LIN {X 0.166,Y -545.979,Z 599.154,A 0.000,B 0.000,C 90.000,E1 63.768} C_DIS
LIN {X 0.022,Y -541.378,Z 599.152,A 0.000,B 0.000,C 90.000,E1 63.435} C_DIS
LIN {X -0.133,Y -535.333,Z 599.150,A 0.000,B 0.000,C 90.000,E1 63.050} C_DIS
LIN {X 0.006,Y -529.277,Z 599.148,A 0.000,B 0.000,C 90.000,E1 62.666} C_DIS
LIN {X 0.118,Y -522.286,Z 599.146,A 0.000,B 0.000,C 90.000,E1 62.281} C_DIS
LIN {X -0.032,Y -515.785,Z 599.144,A 0.000,B 0.000,C 90.000,E1 61.975} C_DIS
LIN {X -0.104,Y -503.976,Z 599.141,A 0.000,B 0.000,C 90.000,E1 61.435} C_DIS
LIN {X -0.129,Y -485.175,Z 599.137,A 0.000,B 0.000,C 90.000,E1 60.589} C_DIS
LIN {X 0.140,Y -461.668,Z 599.130,A 0.000,B 0.000,C 90.000,E1 59.459} C_DIS
LIN {X 0.043,Y -448.327,Z 599.127,A 0.000,B 0.000,C 90.000,E1 58.791} C_DIS
LIN {X 0.001,Y -448.293,Z 599.127,A 0.000,B 0.000,C 90.000,E1 58.791} C_DIS
LIN {X -0.028,Y -444.314,Z 599.115,A 0.000,B 0.000,C 90.000,E1 56.707} C_DIS
LIN {X 0.030,Y -443.665,Z 599.113,A 0.000,B 0.000,C 90.000,E1 56.373} C_DIS
LIN {X 0.020,Y -434.553,Z 599.091,A 0.000,B 0.000,C 90.000,E1 52.431} C_DIS
LIN {X 0.117,Y -431.885,Z 599.083,A 0.000,B 0.000,C 90.000,E1 51.009} C_DIS
LIN {X 0.135,Y -433.279,Z 599.073,A 0.000,B 0.000,C 90.000,E1 49.094} C_DIS
LIN {X -0.208,Y -434.692,Z 599.062,A 0.000,B 0.000,C 90.000,E1 47.148} C_DIS
LIN {X -0.113,Y -435.635,Z 599.054,A 0.000,B 0.000,C 90.000,E1 45.810} C_DIS
LIN {X 0.205,Y -437.080,Z 599.043,A 0.000,B 0.000,C 90.000,E1 43.785} C_DIS
LIN {X 0.041,Y -437.949,Z 599.036,A 0.000,B 0.000,C 90.000,E1 42.486} C_DIS
LIN {X 0.186,Y -438.656,Z 599.029,A 0.000,B 0.000,C 90.000,E1 41.148} C_DIS
LIN {X 0.045,Y -439.277,Z 599.021,A 0.000,B 0.000,C 90.000,E1 39.850} C_DIS
LIN {X -0.061,Y -440.083,Z 599.010,A 0.000,B 0.000,C 90.000,E1 37.890} C_DIS
LIN {X -0.150,Y -440.627,Z 599.000,A 0.000,B 0.000,C 90.000,E1 35.931} C_DIS
LIN {X -0.066,Y -440.906,Z 598.990,A 0.000,B 0.000,C 90.000,E1 34.278} C_DIS
LIN {X -0.016,Y -441.048,Z 598.983,A 0.000,B 0.000,C 90.000,E1 32.959} C_DIS
LIN {X -0.206,Y -441.187,Z 598.976,A 0.000,B 0.000,C 90.000,E1 31.671} C_DIS
LIN {X 0.123,Y -441.488,Z 598.963,A 0.000,B 0.000,C 90.000,E1 29.333} C_DIS
LIN {X 0.016,Y -441.716,Z 598.950,A 0.000,B 0.000,C 90.000,E1 27.052} C_DIS
LIN {X 0.027,Y -441.984,Z 598.941,A 0.000,B 0.000,C 90.000,E1 25.412} C_DIS
LIN {X 0.052,Y -442.349,Z 598.932,A 0.000,B 0.000,C 90.000,E1 23.770} C_DIS
LIN {X -0.240,Y -442.753,Z 598.921,A 0.000,B 0.000,C 90.000,E1 21.844} C_DIS
LIN {X 0.023,Y -443.189,Z 598.912,A 0.000,B 0.000,C 90.000,E1 20.174} C_DIS
LIN {X 0.117,Y -443.894,Z 598.899,A 0.000,B 0.000,C 90.000,E1 17.873} C_DIS
LIN {X 0.242,Y -444.845,Z 598.885,A 0.000,B 0.000,C 90.000,E1 15.245} C_DIS
LIN {X 0.167,Y -446.065,Z 598.870,A 0.000,B 0.000,C 90.000,E1 12.647} C_DIS
LIN {X -0.067,Y -447.666,Z 598.856,A 0.000,B 0.000,C 90.000,E1 10.074} C_DIS
LIN {X -0.092,Y -448.788,Z 598.847,A 0.000,B 0.000,C 90.000,E1 8.454} C_DIS
LIN {X 0.101,Y -450.355,Z 598.836,A 0.000,B 0.000,C 90.000,E1 6.486} C_DIS
LIN {X 0.127,Y -452.695,Z 598.822,A 0.000,B 0.000,C 90.000,E1 3.898} C_DIS
LIN {X -0.197,Y -454.692,Z 598.811,A 0.000,B 0.000,C 90.000,E1 2.007} C_DIS
LIN {X -0.174,Y -458.491,Z 598.794,A 0.000,B 0.000,C 90.000,E1 358.854} C_DIS
LIN {X -0.200,Y -462.594,Z 598.778,A 0.000,B 0.000,C 90.000,E1 355.988} C_DIS
LIN {X 0.016,Y -465.061,Z 598.769,A 0.000,B 0.000,C 90.000,E1 354.375} C_DIS
LIN {X -0.162,Y -468.518,Z 598.757,A 0.000,B 0.000,C 90.000,E1 352.186} C_DIS
LIN {X 0.021,Y -470.459,Z 598.750,A 0.000,B 0.000,C 90.000,E1 350.905} C_DIS
LIN {X -0.186,Y -473.399,Z 598.739,A 0.000,B 0.000,C 90.000,E1 349.050} C_DIS
LIN {X 0.155,Y -477.086,Z 598.727,A 0.000,B 0.000,C 90.000,E1 346.825} C_DIS
LIN {X -0.079,Y -480.404,Z 598.717,A 0.000,B 0.000,C 90.000,E1 344.991} C_DIS
LIN {X -0.101,Y -483.276,Z 598.708,A 0.000,B 0.000,C 90.000,E1 343.449} C_DIS
LIN {X 0.073,Y -486.739,Z 598.698,A 0.000,B 0.000,C 90.000,E1 341.583} C_DIS
LIN {X -0.021,Y -489.139,Z 598.691,A 0.000,B 0.000,C 90.000,E1 340.369} C_DIS
LIN {X -0.049,Y -492.084,Z 598.682,A 0.000,B 0.000,C 90.000,E1 338.847} C_DIS
LIN {X 0.151,Y -494.806,Z 598.674,A 0.000,B 0.000,C 90.000,E1 337.305} C_DIS
LIN {X 0.145,Y -497.417,Z 598.666,A 0.000,B 0.000,C 90.000,E1 335.793} C_DIS
LIN {X -0.200,Y -500.222,Z 598.656,A 0.000,B 0.000,C 90.000,E1 334.024} C_DIS
LIN {X 0.050,Y -502.104,Z 598.649,A 0.000,B 0.000,C 90.000,E1 332.794} C_DIS
LIN {X -0.111,Y -505.249,Z 598.637,A 0.000,B 0.000,C 90.000,E1 330.717} C_DIS
LIN {X 0.042,Y -508.368,Z 598.626,A 0.000,B 0.000,C 90.000,E1 328.614} C_DIS
LIN {X -0.057,Y -511.830,Z 598.614,A 0.000,B 0.000,C 90.000,E1 326.548} C_DIS
LIN {X -0.129,Y -516.286,Z 598.601,A 0.000,B 0.000,C 90.000,E1 324.196} C_DIS
LIN {X -0.095,Y -519.677,Z 598.591,A 0.000,B 0.000,C 90.000,E1 322.431} C_DIS
LIN {X 0.243,Y -523.373,Z 598.582,A 0.000,B 0.000,C 90.000,E1 320.642} C_DIS
LIN {X 0.111,Y -525.794,Z 598.577,A 0.000,B 0.000,C 90.000,E1 319.784} C_DIS
LIN {X 0.011,Y -526.732,Z 598.575,A 0.000,B 0.000,C 90.000,E1 319.504} C_DIS
LIN {X 0.085,Y -529.285,Z 598.572,A 0.000,B 0.000,C 90.000,E1 318.933} C_DIS
LIN {X 0.244,Y -529.830,Z 598.571,A 0.000,B 0.000,C 90.000,E1 318.771} C_DIS
LIN {X 0.215,Y -531.524,Z 598.570,A 0.000,B 0.000,C 90.000,E1 318.485} C_DIS
LIN {X -0.144,Y -534.100,Z 598.568,A 0.000,B 0.000,C 90.000,E1 318.243} C_DIS
LIN {X -0.100,Y -536.720,Z 598.566,A 0.000,B 0.000,C 90.000,E1 317.957} C_DIS
LIN {X -0.059,Y -539.484,Z 598.565,A 0.000,B 0.000,C 90.000,E1 317.676} C_DIS
LIN {X -0.062,Y -544.568,Z 598.562,A 0.000,B 0.000,C 90.000,E1 317.229} C_DIS
LIN {X 0.172,Y -566.738,Z 598.553,A 0.000,B 0.000,C 90.000,E1 315.486} C_DIS
LIN {X -0.044,Y -584.428,Z 598.546,A 0.000,B 0.000,C 90.000,E1 314.190} C_DIS
LIN {X -0.296,Y -590.237,Z 598.543,A 0.000,B 0.000,C 90.000,E1 313.785} C_DIS
LIN {X -0.116,Y -598.732,Z 598.539,A 0.000,B 0.000,C 90.000,E1 313.095} C_DIS
LIN {X 0.176,Y -604.081,Z 598.537,A 0.000,B 0.000,C 90.000,E1 312.609} C_DIS
LIN {X -0.228,Y -608.017,Z 598.535,A 0.000,B 0.000,C 90.000,E1 312.285} C_DIS
LIN {X -0.022,Y -616.798,Z 598.530,A 0.000,B 0.000,C 90.000,E1 311.391} C_DIS
LIN {X -0.281,Y -624.670,Z 598.525,A 0.000,B 0.000,C 90.000,E1 310.539} C_DIS
LIN {X 0.259,Y -631.210,Z 598.521,A 0.000,B 0.000,C 90.000,E1 309.725} C_DIS
LIN {X 0.001,Y -637.456,Z 598.517,A 0.000,B 0.000,C 90.000,E1 308.991} C_DIS
LIN {X 0.184,Y -644.336,Z 598.512,A 0.000,B 0.000,C 90.000,E1 308.096} C_DIS
LIN {X -0.383,Y -648.858,Z 598.508,A 0.000,B 0.000,C 90.000,E1 307.523} C_DIS
LIN {X -0.030,Y -652.251,Z 598.506,A 0.000,B 0.000,C 90.000,E1 306.996} C_DIS
LIN {X -0.048,Y -655.376,Z 598.503,A 0.000,B 0.000,C 90.000,E1 306.503} C_DIS
LIN {X -0.004,Y -658.863,Z 598.499,A 0.000,B 0.000,C 90.000,E1 305.884} C_DIS
LIN {X 0.077,Y -662.080,Z 598.496,A 0.000,B 0.000,C 90.000,E1 305.264} C_DIS
LIN {X 0.074,Y -663.896,Z 598.494,A 0.000,B 0.000,C 90.000,E1 304.898} C_DIS
LIN {X -0.295,Y -667.172,Z 598.490,A 0.000,B 0.000,C 90.000,E1 304.199} C_DIS
LIN {X -0.080,Y -670.198,Z 598.486,A 0.000,B 0.000,C 90.000,E1 303.452} C_DIS
LIN {X -0.396,Y -672.978,Z 598.482,A 0.000,B 0.000,C 90.000,E1 302.752} C_DIS
LIN {X -0.001,Y -677.459,Z 598.475,A 0.000,B 0.000,C 90.000,E1 301.514} C_DIS
LIN {X -0.040,Y -682.613,Z 598.467,A 0.000,B 0.000,C 90.000,E1 300.079} C_DIS
LIN {X -0.063,Y -685.873,Z 598.462,A 0.000,B 0.000,C 90.000,E1 299.127} C_DIS
LIN {X 0.214,Y -688.976,Z 598.457,A 0.000,B 0.000,C 90.000,E1 298.153} C_DIS
LIN {X 0.217,Y -691.869,Z 598.451,A 0.000,B 0.000,C 90.000,E1 297.206} C_DIS
LIN {X 0.084,Y -693.221,Z 598.449,A 0.000,B 0.000,C 90.000,E1 296.744} C_DIS
LIN {X -0.045,Y -694.071,Z 598.446,A 0.000,B 0.000,C 90.000,E1 296.283} C_DIS
LIN {X -0.102,Y -694.440,Z 598.445,A 0.000,B 0.000,C 90.000,E1 296.052} C_DIS
LIN {X 0.149,Y -694.357,Z 598.443,A 0.000,B 0.000,C 90.000,E1 295.796} C_DIS
LIN {X 0.025,Y -693.740,Z 598.441,A 0.000,B 0.000,C 90.000,E1 295.335} C_DIS
LIN {X 0.273,Y -692.734,Z 598.440,A 0.000,B 0.000,C 90.000,E1 295.079} C_DIS
LIN {X -0.278,Y -690.914,Z 598.438,A 0.000,B 0.000,C 90.000,E1 294.771} C_DIS
LIN {X -0.158,Y -690.215,Z 598.437,A 0.000,B 0.000,C 90.000,E1 294.643} C_DIS
LIN {X -0.039,Y -689.136,Z 598.436,A 0.000,B 0.000,C 90.000,E1 294.515} C_DIS
LIN {X 0.078,Y -687.455,Z 598.436,A 0.000,B 0.000,C 90.000,E1 294.387} C_DIS
LIN {X -0.137,Y -683.985,Z 598.434,A 0.000,B 0.000,C 90.000,E1 294.207} C_DIS
LIN {X -0.111,Y -682.117,Z 598.434,A 0.000,B 0.000,C 90.000,E1 294.079} C_DIS
LIN {X 0.259,Y -680.132,Z 598.433,A 0.000,B 0.000,C 90.000,E1 293.951} C_DIS
LIN {X -0.069,Y -673.321,Z 598.432,A 0.000,B 0.000,C 90.000,E1 293.770} C_DIS
LIN {X 0.235,Y -669.043,Z 598.432,A 0.000,B 0.000,C 90.000,E1 293.643} C_DIS
LIN {X -0.119,Y -659.386,Z 598.431,A 0.000,B 0.000,C 90.000,E1 293.515} C_DIS
LIN {X -0.084,Y -646.367,Z 598.430,A 0.000,B 0.000,C 90.000,E1 293.334} C_DIS
LIN {X -0.034,Y -636.744,Z 598.429,A 0.000,B 0.000,C 90.000,E1 293.153} C_DIS
LIN {X -0.173,Y -627.009,Z 598.427,A 0.000,B 0.000,C 90.000,E1 292.950} C_DIS
LIN {X -0.121,Y -613.924,Z 598.425,A 0.000,B 0.000,C 90.000,E1 292.589} C_DIS
LIN {X 0.130,Y -579.349,Z 598.419,A 0.000,B 0.000,C 90.000,E1 291.482} C_DIS
LIN {X 0.137,Y -569.347,Z 598.418,A 0.000,B 0.000,C 90.000,E1 291.173} C_DIS
LIN {X -0.267,Y -565.886,Z 598.417,A 0.000,B 0.000,C 90.000,E1 291.099} C_DIS
LIN {X -0.154,Y -563.479,Z 598.416,A 0.000,B 0.000,C 90.000,E1 290.972} C_DIS
LIN {X 0.119,Y -560.661,Z 598.416,A 0.000,B 0.000,C 90.000,E1 290.791} C_DIS
LIN {X 0.065,Y -560.619,Z 598.416,A 0.000,B 0.000,C 90.000,E1 290.791} C_DIS
LIN {X -0.201,Y -559.519,Z 598.415,A 0.000,B 0.000,C 90.000,E1 290.663} C_DIS
LIN {X 0.279,Y -559.491,Z 598.415,A 0.000,B 0.000,C 90.000,E1 290.610} C_DIS
LIN {X -0.199,Y -558.876,Z 598.412,A 0.000,B 0.000,C 90.000,E1 290.248} C_DIS
LIN {X 0.055,Y -558.699,Z 598.402,A 0.000,B 0.000,C 90.000,E1 288.362} C_DIS
LIN {X 0.240,Y -558.547,Z 598.397,A 0.000,B 0.000,C 90.000,E1 287.511} C_DIS
LIN {X 0.137,Y -558.104,Z 598.390,A 0.000,B 0.000,C 90.000,E1 286.134} C_DIS
LIN {X 0.279,Y -557.667,Z 598.384,A 0.000,B 0.000,C 90.000,E1 285.009} C_DIS
LIN {X 0.145,Y -556.814,Z 598.374,A 0.000,B 0.000,C 90.000,E1 283.355} C_DIS
LIN {X -0.265,Y -556.046,Z 598.367,A 0.000,B 0.000,C 90.000,E1 282.007} C_DIS
LIN {X 0.115,Y -554.956,Z 598.356,A 0.000,B 0.000,C 90.000,E1 280.018} C_DIS
LIN {X -0.275,Y -553.920,Z 598.345,A 0.000,B 0.000,C 90.000,E1 278.106} C_DIS
LIN {X 0.177,Y -553.280,Z 598.337,A 0.000,B 0.000,C 90.000,E1 276.663} C_DIS
LIN {X 0.118,Y -552.541,Z 598.328,A 0.000,B 0.000,C 90.000,E1 274.992} C_DIS
LIN {X 0.088,Y -551.894,Z 598.317,A 0.000,B 0.000,C 90.000,E1 273.037} C_DIS
LIN {X -0.023,Y -551.381,Z 598.306,A 0.000,B 0.000,C 90.000,E1 271.088} C_DIS
LIN {X -0.271,Y -551.012,Z 598.298,A 0.000,B 0.000,C 90.000,E1 269.714} C_DIS
LIN {X 0.153,Y -550.278,Z 598.287,A 0.000,B 0.000,C 90.000,E1 267.707} C_DIS
LIN {X -0.102,Y -549.713,Z 598.280,A 0.000,B 0.000,C 90.000,E1 266.331} C_DIS
LIN {X 0.215,Y -549.027,Z 598.272,A 0.000,B 0.000,C 90.000,E1 264.894} C_DIS
LIN {X -0.033,Y -548.223,Z 598.264,A 0.000,B 0.000,C 90.000,E1 263.514} C_DIS
LIN {X 0.281,Y -547.287,Z 598.258,A 0.000,B 0.000,C 90.000,E1 262.356} C_DIS
LIN {X 0.058,Y -546.050,Z 598.250,A 0.000,B 0.000,C 90.000,E1 260.971} C_DIS
LIN {X 0.068,Y -544.125,Z 598.239,A 0.000,B 0.000,C 90.000,E1 258.993} C_DIS
LIN {X -0.115,Y -543.093,Z 598.233,A 0.000,B 0.000,C 90.000,E1 257.881} C_DIS
LIN {X -0.033,Y -541.350,Z 598.223,A 0.000,B 0.000,C 90.000,E1 256.172} C_DIS
LIN {X -0.128,Y -540.226,Z 598.217,A 0.000,B 0.000,C 90.000,E1 255.046} C_DIS
LIN {X -0.027,Y -538.775,Z 598.209,A 0.000,B 0.000,C 90.000,E1 253.614} C_DIS
LIN {X 0.045,Y -537.283,Z 598.201,A 0.000,B 0.000,C 90.000,E1 252.181} C_DIS
LIN {X 0.038,Y -536.067,Z 598.195,A 0.000,B 0.000,C 90.000,E1 251.040} C_DIS
LIN {X -0.109,Y -534.119,Z 598.187,A 0.000,B 0.000,C 90.000,E1 249.625} C_DIS
LIN {X 0.213,Y -531.664,Z 598.179,A 0.000,B 0.000,C 90.000,E1 248.156} C_DIS
LIN {X -0.199,Y -529.517,Z 598.172,A 0.000,B 0.000,C 90.000,E1 247.050} C_DIS
LIN {X -0.261,Y -526.695,Z 598.164,A 0.000,B 0.000,C 90.000,E1 245.613} C_DIS
LIN {X -0.155,Y -523.732,Z 598.156,A 0.000,B 0.000,C 90.000,E1 244.152} C_DIS
LIN {X 0.130,Y -520.515,Z 598.148,A 0.000,B 0.000,C 90.000,E1 242.666} C_DIS
LIN {X -0.014,Y -517.839,Z 598.142,A 0.000,B 0.000,C 90.000,E1 241.513} C_DIS
LIN {X 0.044,Y -514.913,Z 598.135,A 0.000,B 0.000,C 90.000,E1 240.333} C_DIS
LIN {X -0.153,Y -509.069,Z 598.122,A 0.000,B 0.000,C 90.000,E1 237.995} C_DIS
LIN {X 0.028,Y -506.047,Z 598.116,A 0.000,B 0.000,C 90.000,E1 236.786} C_DIS
LIN {X 0.018,Y -502.654,Z 598.109,A 0.000,B 0.000,C 90.000,E1 235.595} C_DIS
LIN {X -0.034,Y -499.205,Z 598.102,A 0.000,B 0.000,C 90.000,E1 234.402} C_DIS
LIN {X -0.152,Y -491.971,Z 598.087,A 0.000,B 0.000,C 90.000,E1 231.698} C_DIS
LIN {X 0.068,Y -487.986,Z 598.079,A 0.000,B 0.000,C 90.000,E1 230.150} C_DIS
LIN {X 0.015,Y -484.808,Z 598.072,A 0.000,B 0.000,C 90.000,E1 228.933} C_DIS
LIN {X -0.028,Y -479.413,Z 598.060,A 0.000,B 0.000,C 90.000,E1 226.782} C_DIS
LIN {X -0.009,Y -474.908,Z 598.050,A 0.000,B 0.000,C 90.000,E1 224.919} C_DIS
LIN {X -0.181,Y -471.290,Z 598.041,A 0.000,B 0.000,C 90.000,E1 223.380} C_DIS
LIN {X 0.021,Y -466.931,Z 598.030,A 0.000,B 0.000,C 90.000,E1 221.472} C_DIS
LIN {X -0.034,Y -464.181,Z 598.023,A 0.000,B 0.000,C 90.000,E1 220.216} C_DIS
LIN {X -0.203,Y -459.497,Z 598.011,A 0.000,B 0.000,C 90.000,E1 218.016} C_DIS
LIN {X 0.035,Y -456.868,Z 598.004,A 0.000,B 0.000,C 90.000,E1 216.710} C_DIS
LIN {X 0.052,Y -453.745,Z 597.995,A 0.000,B 0.000,C 90.000,E1 215.105} C_DIS
LIN {X -0.116,Y -448.841,Z 597.981,A 0.000,B 0.000,C 90.000,E1 212.546} C_DIS
LIN {X -0.054,Y -445.372,Z 597.970,A 0.000,B 0.000,C 90.000,E1 210.590} C_DIS
LIN {X 0.079,Y -441.814,Z 597.959,A 0.000,B 0.000,C 90.000,E1 208.615} C_DIS
LIN {X -0.084,Y -438.365,Z 597.948,A 0.000,B 0.000,C 90.000,E1 206.668} C_DIS
LIN {X -0.149,Y -435.482,Z 597.939,A 0.000,B 0.000,C 90.000,E1 205.027} C_DIS
LIN {X -0.047,Y -432.098,Z 597.928,A 0.000,B 0.000,C 90.000,E1 203.025} C_DIS
LIN {X 0.000,Y -429.390,Z 597.919,A 0.000,B 0.000,C 90.000,E1 201.354} C_DIS
LIN {X -0.162,Y -425.683,Z 597.906,A 0.000,B 0.000,C 90.000,E1 199.033} C_DIS
LIN {X 0.056,Y -422.755,Z 597.894,A 0.000,B 0.000,C 90.000,E1 196.985} C_DIS
LIN {X 0.075,Y -419.965,Z 597.883,A 0.000,B 0.000,C 90.000,E1 194.954} C_DIS
LIN {X 0.111,Y -418.085,Z 597.876,A 0.000,B 0.000,C 90.000,E1 193.592} C_DIS
LIN {X 0.204,Y -415.072,Z 597.864,A 0.000,B 0.000,C 90.000,E1 191.535} C_DIS
LIN {X 0.176,Y -410.918,Z 597.847,A 0.000,B 0.000,C 90.000,E1 188.454} C_DIS
LIN {X -0.144,Y -408.830,Z 597.838,A 0.000,B 0.000,C 90.000,E1 186.777} C_DIS
LIN {X -0.168,Y -405.709,Z 597.824,A 0.000,B 0.000,C 90.000,E1 184.359} C_DIS
LIN {X -0.135,Y -401.282,Z 597.799,A 0.000,B 0.000,C 90.000,E1 179.828} C_DIS
LIN {X -0.112,Y -399.169,Z 597.781,A 0.000,B 0.000,C 90.000,E1 176.674} C_DIS
LIN {X -0.051,Y -398.035,Z 597.766,A 0.000,B 0.000,C 90.000,E1 173.856} C_DIS
LIN {X 0.078,Y -397.457,Z 597.752,A 0.000,B 0.000,C 90.000,E1 171.376} C_DIS
LIN {X -0.044,Y -397.250,Z 597.737,A 0.000,B 0.000,C 90.000,E1 168.578} C_DIS
LIN {X 0.002,Y -397.566,Z 597.721,A 0.000,B 0.000,C 90.000,E1 165.755} C_DIS
LIN {X 0.104,Y -398.040,Z 597.709,A 0.000,B 0.000,C 90.000,E1 163.630} C_DIS
LIN {X 0.099,Y -398.630,Z 597.699,A 0.000,B 0.000,C 90.000,E1 161.873} C_DIS
LIN {X -0.099,Y -399.432,Z 597.686,A 0.000,B 0.000,C 90.000,E1 159.444} C_DIS
LIN {X -0.225,Y -400.269,Z 597.674,A 0.000,B 0.000,C 90.000,E1 157.358} C_DIS
LIN {X -0.026,Y -401.172,Z 597.662,A 0.000,B 0.000,C 90.000,E1 155.229} C_DIS
LIN {X 0.114,Y -401.924,Z 597.653,A 0.000,B 0.000,C 90.000,E1 153.461} C_DIS
LIN {X -0.161,Y -402.572,Z 597.645,A 0.000,B 0.000,C 90.000,E1 152.103} C_DIS
LIN {X -0.086,Y -403.408,Z 597.633,A 0.000,B 0.000,C 90.000,E1 149.999} C_DIS
LIN {X -0.033,Y -403.993,Z 597.624,A 0.000,B 0.000,C 90.000,E1 148.250} C_DIS
LIN {X 0.030,Y -404.457,Z 597.614,A 0.000,B 0.000,C 90.000,E1 146.501} C_DIS
LIN {X 0.111,Y -404.966,Z 597.602,A 0.000,B 0.000,C 90.000,E1 144.402} C_DIS
LIN {X -0.126,Y -405.515,Z 597.591,A 0.000,B 0.000,C 90.000,E1 142.351} C_DIS
LIN {X -0.175,Y -406.136,Z 597.579,A 0.000,B 0.000,C 90.000,E1 140.275} C_DIS
LIN {X 0.053,Y -406.672,Z 597.568,A 0.000,B 0.000,C 90.000,E1 138.162} C_DIS
LIN {X 0.005,Y -406.892,Z 597.560,A 0.000,B 0.000,C 90.000,E1 136.782} C_DIS
LIN {X 0.204,Y -407.210,Z 597.548,A 0.000,B 0.000,C 90.000,E1 134.676} C_DIS
LIN {X -0.011,Y -407.436,Z 597.539,A 0.000,B 0.000,C 90.000,E1 132.975} C_DIS
LIN {X -0.065,Y -407.624,Z 597.527,A 0.000,B 0.000,C 90.000,E1 130.906} C_DIS
LIN {X -0.215,Y -407.826,Z 597.518,A 0.000,B 0.000,C 90.000,E1 129.197} C_DIS
LIN {X -0.151,Y -407.834,Z 597.515,A 0.000,B 0.000,C 90.000,E1 128.669} C_DIS
LIN {X -0.201,Y -415.250,Z 597.500,A 0.000,B 0.000,C 90.000,E1 126.091} C_DIS
LIN {X -0.091,Y -416.909,Z 597.497,A 0.000,B 0.000,C 90.000,E1 125.391} C_DIS
LIN {X 0.101,Y -425.710,Z 597.478,A 0.000,B 0.000,C 90.000,E1 121.957} C_DIS
LIN {X 0.062,Y -425.748,Z 597.478,A 0.000,B 0.000,C 90.000,E1 121.957} C_DIS
LIN {X 0.143,Y -435.597,Z 597.475,A 0.000,B 0.000,C 90.000,E1 121.465} C_DIS
LIN {X -0.037,Y -442.412,Z 597.473,A 0.000,B 0.000,C 90.000,E1 121.180} C_DIS
LIN {X -0.064,Y -449.171,Z 597.471,A 0.000,B 0.000,C 90.000,E1 120.846} C_DIS
LIN {X 0.070,Y -452.676,Z 597.470,A 0.000,B 0.000,C 90.000,E1 120.669} C_DIS
LIN {X 0.030,Y -466.023,Z 597.467,A 0.000,B 0.000,C 90.000,E1 120.001} C_DIS
LIN {X 0.058,Y -475.942,Z 597.464,A 0.000,B 0.000,C 90.000,E1 119.461} C_DIS
LIN {X 0.201,Y -482.620,Z 597.462,A 0.000,B 0.000,C 90.000,E1 119.077} C_DIS
LIN {X -0.146,Y -493.965,Z 597.458,A 0.000,B 0.000,C 90.000,E1 118.437} C_DIS
LIN {X -0.083,Y -500.278,Z 597.456,A 0.000,B 0.000,C 90.000,E1 118.025} C_DIS
LIN {X 0.037,Y -509.700,Z 597.452,A 0.000,B 0.000,C 90.000,E1 117.385} C_DIS
LIN {X -0.148,Y -519.934,Z 597.448,A 0.000,B 0.000,C 90.000,E1 116.668} C_DIS
LIN {X -0.032,Y -527.143,Z 597.445,A 0.000,B 0.000,C 90.000,E1 116.104} C_DIS
LIN {X -0.109,Y -532.984,Z 597.442,A 0.000,B 0.000,C 90.000,E1 115.643} C_DIS
LIN {X 0.040,Y -540.321,Z 597.439,A 0.000,B 0.000,C 90.000,E1 115.027} C_DIS
LIN {X 0.195,Y -545.812,Z 597.436,A 0.000,B 0.000,C 90.000,E1 114.515} C_DIS
LIN {X -0.133,Y -550.789,Z 597.434,A 0.000,B 0.000,C 90.000,E1 114.079} C_DIS
LIN {X -0.126,Y -555.397,Z 597.431,A 0.000,B 0.000,C 90.000,E1 113.567} C_DIS
LIN {X 0.171,Y -561.281,Z 597.427,A 0.000,B 0.000,C 90.000,E1 112.823} C_DIS
LIN {X -0.257,Y -563.091,Z 597.425,A 0.000,B 0.000,C 90.000,E1 112.589} C_DIS
LIN {X -0.168,Y -565.816,Z 597.423,A 0.000,B 0.000,C 90.000,E1 112.206} C_DIS
LIN {X -0.336,Y -570.004,Z 597.419,A 0.000,B 0.000,C 90.000,E1 111.535} C_DIS
LIN {X 0.190,Y -574.425,Z 597.415,A 0.000,B 0.000,C 90.000,E1 110.663} C_DIS
LIN {X -0.178,Y -578.433,Z 597.410,A 0.000,B 0.000,C 90.000,E1 109.885} C_DIS
LIN {X 0.042,Y -580.900,Z 597.407,A 0.000,B 0.000,C 90.000,E1 109.322} C_DIS
LIN {X -0.259,Y -584.375,Z 597.403,A 0.000,B 0.000,C 90.000,E1 108.544} C_DIS
LIN {X -0.194,Y -586.556,Z 597.400,A 0.000,B 0.000,C 90.000,E1 108.000} C_DIS
LIN {X -0.021,Y -590.310,Z 597.394,A 0.000,B 0.000,C 90.000,E1 106.913} C_DIS
LIN {X -0.229,Y -592.947,Z 597.390,A 0.000,B 0.000,C 90.000,E1 106.134} C_DIS
LIN {X 0.138,Y -597.029,Z 597.382,A 0.000,B 0.000,C 90.000,E1 104.773} C_DIS
LIN {X 0.301,Y -602.058,Z 597.373,A 0.000,B 0.000,C 90.000,E1 103.175} C_DIS
LIN {X 0.041,Y -607.979,Z 597.363,A 0.000,B 0.000,C 90.000,E1 101.366} C_DIS
LIN {X -0.064,Y -612.191,Z 597.356,A 0.000,B 0.000,C 90.000,E1 100.074} C_DIS
LIN {X -0.315,Y -616.167,Z 597.349,A 0.000,B 0.000,C 90.000,E1 98.803} C_DIS
LIN {X 0.124,Y -619.932,Z 597.342,A 0.000,B 0.000,C 90.000,E1 97.473} C_DIS
LIN {X 0.011,Y -623.481,Z 597.335,A 0.000,B 0.000,C 90.000,E1 96.201} C_DIS
LIN {X -0.148,Y -625.431,Z 597.330,A 0.000,B 0.000,C 90.000,E1 95.448} C_DIS
LIN {X 0.273,Y -627.230,Z 597.326,A 0.000,B 0.000,C 90.000,E1 94.645} C_DIS
LIN {X 0.090,Y -628.750,Z 597.322,A 0.000,B 0.000,C 90.000,E1 93.898} C_DIS
LIN {X 0.273,Y -630.629,Z 597.316,A 0.000,B 0.000,C 90.000,E1 92.865} C_DIS
LIN {X 0.213,Y -632.546,Z 597.309,A 0.000,B 0.000,C 90.000,E1 91.604} C_DIS
LIN {X 0.056,Y -633.540,Z 597.305,A 0.000,B 0.000,C 90.000,E1 90.859} C_DIS
LIN {X -0.090,Y -634.288,Z 597.301,A 0.000,B 0.000,C 90.000,E1 90.115} C_DIS
LIN {X -0.226,Y -634.788,Z 597.296,A 0.000,B 0.000,C 90.000,E1 89.370} C_DIS
LIN {X 0.274,Y -635.067,Z 597.292,A 0.000,B 0.000,C 90.000,E1 88.568} C_DIS
LIN {X 0.162,Y -635.153,Z 597.288,A 0.000,B 0.000,C 90.000,E1 87.822} C_DIS
LIN {X -0.199,Y -634.893,Z 597.282,A 0.000,B 0.000,C 90.000,E1 86.846} C_DIS
LIN {X 0.288,Y -634.496,Z 597.278,A 0.000,B 0.000,C 90.000,E1 86.045} C_DIS
LIN {X -0.039,Y -633.735,Z 597.273,A 0.000,B 0.000,C 90.000,E1 85.065} C_DIS
LIN {X -0.008,Y -632.447,Z 597.266,A 0.000,B 0.000,C 90.000,E1 83.799} C_DIS
LIN {X 0.138,Y -631.854,Z 597.263,A 0.000,B 0.000,C 90.000,E1 83.280} C_DIS
LIN {X -0.010,Y -630.674,Z 597.259,A 0.000,B 0.000,C 90.000,E1 82.534} C_DIS
LIN {X -0.294,Y -628.902,Z 597.253,A 0.000,B 0.000,C 90.000,E1 81.546} C_DIS
LIN {X 0.234,Y -627.372,Z 597.249,A 0.000,B 0.000,C 90.000,E1 80.735} C_DIS
LIN {X 0.320,Y -624.623,Z 597.242,A 0.000,B 0.000,C 90.000,E1 79.454} C_DIS
LIN {X -0.254,Y -621.558,Z 597.235,A 0.000,B 0.000,C 90.000,E1 78.229} C_DIS
LIN {X 0.082,Y -618.908,Z 597.229,A 0.000,B 0.000,C 90.000,E1 77.173} C_DIS
LIN {X -0.222,Y -616.052,Z 597.223,A 0.000,B 0.000,C 90.000,E1 76.172} C_DIS
LIN {X -0.056,Y -612.192,Z 597.216,A 0.000,B 0.000,C 90.000,E1 74.866} C_DIS
LIN {X -0.204,Y -609.669,Z 597.212,A 0.000,B 0.000,C 90.000,E1 74.102} C_DIS
LIN {X -0.214,Y -606.897,Z 597.207,A 0.000,B 0.000,C 90.000,E1 73.323} C_DIS
LIN {X -0.251,Y -603.838,Z 597.203,A 0.000,B 0.000,C 90.000,E1 72.543} C_DIS
LIN {X -0.319,Y -600.529,Z 597.199,A 0.000,B 0.000,C 90.000,E1 71.764} C_DIS
LIN {X -0.180,Y -597.576,Z 597.195,A 0.000,B 0.000,C 90.000,E1 71.094} C_DIS
LIN {X -0.122,Y -593.748,Z 597.190,A 0.000,B 0.000,C 90.000,E1 70.296} C_DIS
LIN {X -0.043,Y -590.353,Z 597.187,A 0.000,B 0.000,C 90.000,E1 69.625} C_DIS
LIN {X 0.004,Y -586.670,Z 597.183,A 0.000,B 0.000,C 90.000,E1 68.954} C_DIS
LIN {X 0.055,Y -582.749,Z 597.179,A 0.000,B 0.000,C 90.000,E1 68.284} C_DIS
LIN {X -0.263,Y -579.534,Z 597.177,A 0.000,B 0.000,C 90.000,E1 67.794} C_DIS
LIN {X 0.086,Y -574.070,Z 597.172,A 0.000,B 0.000,C 90.000,E1 66.975} C_DIS
LIN {X -0.201,Y -570.192,Z 597.169,A 0.000,B 0.000,C 90.000,E1 66.485} C_DIS
LIN {X 0.253,Y -564.781,Z 597.166,A 0.000,B 0.000,C 90.000,E1 65.793} C_DIS
LIN {X 0.097,Y -560.305,Z 597.163,A 0.000,B 0.000,C 90.000,E1 65.305} C_DIS
LIN {X -0.252,Y -555.562,Z 597.160,A 0.000,B 0.000,C 90.000,E1 64.845} C_DIS
LIN {X 0.046,Y -550.417,Z 597.157,A 0.000,B 0.000,C 90.000,E1 64.332} C_DIS
LIN {X -0.183,Y -544.861,Z 597.155,A 0.000,B 0.000,C 90.000,E1 63.896} C_DIS
LIN {X -0.032,Y -539.093,Z 597.153,A 0.000,B 0.000,C 90.000,E1 63.461} C_DIS
LIN {X 0.178,Y -534.164,Z 597.151,A 0.000,B 0.000,C 90.000,E1 63.127} C_DIS
LIN {X 0.192,Y -527.618,Z 597.149,A 0.000,B 0.000,C 90.000,E1 62.743} C_DIS
LIN {X -0.099,Y -520.593,Z 597.147,A 0.000,B 0.000,C 90.000,E1 62.410} C_DIS
LIN {X -0.050,Y -515.458,Z 597.145,A 0.000,B 0.000,C 90.000,E1 62.153} C_DIS
LIN {X 0.023,Y -503.311,Z 597.142,A 0.000,B 0.000,C 90.000,E1 61.591} C_DIS
LIN {X 0.072,Y -482.856,Z 597.137,A 0.000,B 0.000,C 90.000,E1 60.667} C_DIS
LIN {X -0.103,Y -462.472,Z 597.132,A 0.000,B 0.000,C 90.000,E1 59.744} C_DIS
LIN {X -0.278,Y -448.859,Z 597.128,A 0.000,B 0.000,C 90.000,E1 59.076} C_DIS
LIN {X 0.295,Y -448.803,Z 597.128,A 0.000,B 0.000,C 90.000,E1 58.997} C_DIS
LIN {X 0.138,Y -444.131,Z 597.115,A 0.000,B 0.000,C 90.000,E1 56.580} C_DIS
LIN {X 0.128,Y -442.543,Z 597.111,A 0.000,B 0.000,C 90.000,E1 55.928} C_DIS
LIN {X 0.084,Y -433.691,Z 597.089,A 0.000,B 0.000,C 90.000,E1 51.984} C_DIS
LIN {X -0.012,Y -432.290,Z 597.085,A 0.000,B 0.000,C 90.000,E1 51.251} C_DIS
LIN {X 0.190,Y -432.649,Z 597.082,A 0.000,B 0.000,C 90.000,E1 50.642} C_DIS
LIN {X -0.058,Y -433.941,Z 597.072,A 0.000,B 0.000,C 90.000,E1 49.013} C_DIS
LIN {X 0.286,Y -435.162,Z 597.063,A 0.000,B 0.000,C 90.000,E1 47.310} C_DIS
LIN {X -0.228,Y -436.185,Z 597.056,A 0.000,B 0.000,C 90.000,E1 46.053} C_DIS
LIN {X 0.057,Y -437.911,Z 597.043,A 0.000,B 0.000,C 90.000,E1 43.704} C_DIS
LIN {X 0.201,Y -438.752,Z 597.036,A 0.000,B 0.000,C 90.000,E1 42.366} C_DIS
LIN {X 0.063,Y -439.459,Z 597.028,A 0.000,B 0.000,C 90.000,E1 41.067} C_DIS
LIN {X -0.068,Y -440.051,Z 597.021,A 0.000,B 0.000,C 90.000,E1 39.769} C_DIS
LIN {X -0.158,Y -440.829,Z 597.010,A 0.000,B 0.000,C 90.000,E1 37.810} C_DIS
LIN {X -0.172,Y -441.252,Z 597.001,A 0.000,B 0.000,C 90.000,E1 36.171} C_DIS
LIN {X -0.182,Y -441.548,Z 596.992,A 0.000,B 0.000,C 90.000,E1 34.532} C_DIS
LIN {X -0.126,Y -441.643,Z 596.984,A 0.000,B 0.000,C 90.000,E1 33.214} C_DIS
LIN {X 0.113,Y -441.805,Z 596.975,A 0.000,B 0.000,C 90.000,E1 31.544} C_DIS
LIN {X 0.028,Y -441.995,Z 596.964,A 0.000,B 0.000,C 90.000,E1 29.589} C_DIS
LIN {X -0.067,Y -442.208,Z 596.952,A 0.000,B 0.000,C 90.000,E1 27.308} C_DIS
LIN {X -0.009,Y -442.480,Z 596.941,A 0.000,B 0.000,C 90.000,E1 25.335} C_DIS
LIN {X 0.019,Y -442.801,Z 596.932,A 0.000,B 0.000,C 90.000,E1 23.695} C_DIS
LIN {X -0.125,Y -443.125,Z 596.923,A 0.000,B 0.000,C 90.000,E1 22.078} C_DIS
LIN {X -0.015,Y -443.531,Z 596.914,A 0.000,B 0.000,C 90.000,E1 20.429} C_DIS
LIN {X -0.048,Y -444.240,Z 596.899,A 0.000,B 0.000,C 90.000,E1 17.819} C_DIS
LIN {X -0.183,Y -445.047,Z 596.886,A 0.000,B 0.000,C 90.000,E1 15.552} C_DIS
LIN {X -0.140,Y -446.219,Z 596.872,A 0.000,B 0.000,C 90.000,E1 12.939} C_DIS
LIN {X 0.068,Y -447.747,Z 596.857,A 0.000,B 0.000,C 90.000,E1 10.310} C_DIS
LIN {X 0.117,Y -448.854,Z 596.848,A 0.000,B 0.000,C 90.000,E1 8.681} C_DIS
LIN {X -0.004,Y -450.610,Z 596.836,A 0.000,B 0.000,C 90.000,E1 6.429} C_DIS
LIN {X -0.163,Y -452.637,Z 596.823,A 0.000,B 0.000,C 90.000,E1 4.188} C_DIS
LIN {X 0.168,Y -454.933,Z 596.811,A 0.000,B 0.000,C 90.000,E1 1.892} C_DIS
LIN {X -0.173,Y -458.635,Z 596.794,A 0.000,B 0.000,C 90.000,E1 358.854} C_DIS
LIN {X 0.066,Y -462.209,Z 596.779,A 0.000,B 0.000,C 90.000,E1 356.274} C_DIS
LIN {X 0.025,Y -465.161,Z 596.769,A 0.000,B 0.000,C 90.000,E1 354.375} C_DIS
LIN {X -0.150,Y -468.599,Z 596.757,A 0.000,B 0.000,C 90.000,E1 352.186} C_DIS
LIN {X -0.223,Y -471.028,Z 596.748,A 0.000,B 0.000,C 90.000,E1 350.622} C_DIS
LIN {X 0.125,Y -473.982,Z 596.737,A 0.000,B 0.000,C 90.000,E1 348.701} C_DIS
LIN {X 0.013,Y -477.675,Z 596.725,A 0.000,B 0.000,C 90.000,E1 346.533} C_DIS
LIN {X 0.229,Y -481.596,Z 596.713,A 0.000,B 0.000,C 90.000,E1 344.338} C_DIS
LIN {X -0.092,Y -484.451,Z 596.705,A 0.000,B 0.000,C 90.000,E1 342.834} C_DIS
LIN {X -0.021,Y -488.593,Z 596.693,A 0.000,B 0.000,C 90.000,E1 340.678} C_DIS
LIN {X -0.028,Y -492.123,Z 596.682,A 0.000,B 0.000,C 90.000,E1 338.847} C_DIS
LIN {X -0.283,Y -494.834,Z 596.674,A 0.000,B 0.000,C 90.000,E1 337.358} C_DIS
LIN {X 0.167,Y -497.455,Z 596.666,A 0.000,B 0.000,C 90.000,E1 335.793} C_DIS
LIN {X 0.214,Y -499.812,Z 596.657,A 0.000,B 0.000,C 90.000,E1 334.280} C_DIS
LIN {X 0.076,Y -502.166,Z 596.649,A 0.000,B 0.000,C 90.000,E1 332.794} C_DIS
LIN {X -0.084,Y -505.338,Z 596.637,A 0.000,B 0.000,C 90.000,E1 330.717} C_DIS
LIN {X 0.072,Y -508.482,Z 596.626,A 0.000,B 0.000,C 90.000,E1 328.614} C_DIS
LIN {X -0.024,Y -511.939,Z 596.614,A 0.000,B 0.000,C 90.000,E1 326.548} C_DIS
LIN {X -0.093,Y -516.339,Z 596.601,A 0.000,B 0.000,C 90.000,E1 324.196} C_DIS
LIN {X 0.001,Y -519.170,Z 596.593,A 0.000,B 0.000,C 90.000,E1 322.718} C_DIS
LIN {X 0.235,Y -523.935,Z 596.580,A 0.000,B 0.000,C 90.000,E1 320.356} C_DIS
LIN {X -0.144,Y -526.680,Z 596.574,A 0.000,B 0.000,C 90.000,E1 319.380} C_DIS
LIN {X 0.009,Y -527.374,Z 596.573,A 0.000,B 0.000,C 90.000,E1 319.218} C_DIS
LIN {X 0.131,Y -528.923,Z 596.571,A 0.000,B 0.000,C 90.000,E1 318.771} C_DIS
LIN {X 0.118,Y -531.315,Z 596.569,A 0.000,B 0.000,C 90.000,E1 318.324} C_DIS
LIN {X 0.282,Y -532.253,Z 596.568,A 0.000,B 0.000,C 90.000,E1 318.162} C_DIS
LIN {X 0.060,Y -535.532,Z 596.565,A 0.000,B 0.000,C 90.000,E1 317.757} C_DIS
LIN {X -0.025,Y -538.642,Z 596.564,A 0.000,B 0.000,C 90.000,E1 317.433} C_DIS
LIN {X -0.138,Y -544.246,Z 596.561,A 0.000,B 0.000,C 90.000,E1 316.944} C_DIS
LIN {X -0.252,Y -554.487,Z 596.556,A 0.000,B 0.000,C 90.000,E1 316.134} C_DIS
LIN {X -0.275,Y -566.353,Z 596.551,A 0.000,B 0.000,C 90.000,E1 315.243} C_DIS
LIN {X 0.289,Y -584.096,Z 596.544,A 0.000,B 0.000,C 90.000,E1 313.866} C_DIS
LIN {X -0.139,Y -592.808,Z 596.540,A 0.000,B 0.000,C 90.000,E1 313.257} C_DIS
LIN {X 0.308,Y -598.401,Z 596.538,A 0.000,B 0.000,C 90.000,E1 312.771} C_DIS
LIN {X 0.132,Y -602.476,Z 596.536,A 0.000,B 0.000,C 90.000,E1 312.447} C_DIS
LIN {X -0.173,Y -606.439,Z 596.534,A 0.000,B 0.000,C 90.000,E1 312.123} C_DIS
LIN {X 0.225,Y -615.269,Z 596.529,A 0.000,B 0.000,C 90.000,E1 311.229} C_DIS
LIN {X 0.286,Y -622.377,Z 596.525,A 0.000,B 0.000,C 90.000,E1 310.458} C_DIS
LIN {X -0.051,Y -627.992,Z 596.521,A 0.000,B 0.000,C 90.000,E1 309.850} C_DIS
LIN {X 0.019,Y -635.456,Z 596.516,A 0.000,B 0.000,C 90.000,E1 308.955} C_DIS
LIN {X 0.175,Y -643.384,Z 596.511,A 0.000,B 0.000,C 90.000,E1 307.935} C_DIS
LIN {X 0.113,Y -647.951,Z 596.507,A 0.000,B 0.000,C 90.000,E1 307.317} C_DIS
LIN {X -0.034,Y -652.174,Z 596.504,A 0.000,B 0.000,C 90.000,E1 306.710} C_DIS
LIN {X -0.086,Y -654.505,Z 596.502,A 0.000,B 0.000,C 90.000,E1 306.343} C_DIS
LIN {X -0.050,Y -658.052,Z 596.498,A 0.000,B 0.000,C 90.000,E1 305.724} C_DIS
LIN {X -0.028,Y -660.685,Z 596.496,A 0.000,B 0.000,C 90.000,E1 305.231} C_DIS
LIN {X 0.066,Y -663.696,Z 596.492,A 0.000,B 0.000,C 90.000,E1 304.612} C_DIS
LIN {X -0.309,Y -666.980,Z 596.488,A 0.000,B 0.000,C 90.000,E1 303.913} C_DIS
LIN {X -0.098,Y -669.977,Z 596.484,A 0.000,B 0.000,C 90.000,E1 303.166} C_DIS
LIN {X -0.005,Y -671.896,Z 596.482,A 0.000,B 0.000,C 90.000,E1 302.673} C_DIS
LIN {X -0.152,Y -675.565,Z 596.476,A 0.000,B 0.000,C 90.000,E1 301.720} C_DIS
LIN {X -0.074,Y -679.971,Z 596.470,A 0.000,B 0.000,C 90.000,E1 300.512} C_DIS
LIN {X 0.121,Y -683.387,Z 596.464,A 0.000,B 0.000,C 90.000,E1 299.539} C_DIS
LIN {X -0.233,Y -686.586,Z 596.459,A 0.000,B 0.000,C 90.000,E1 298.615} C_DIS
LIN {X 0.056,Y -689.582,Z 596.454,A 0.000,B 0.000,C 90.000,E1 297.641} C_DIS
LIN {X 0.144,Y -691.708,Z 596.450,A 0.000,B 0.000,C 90.000,E1 296.924} C_DIS
LIN {X -0.305,Y -692.811,Z 596.447,A 0.000,B 0.000,C 90.000,E1 296.488} C_DIS
LIN {X -0.061,Y -693.216,Z 596.446,A 0.000,B 0.000,C 90.000,E1 296.232} C_DIS
LIN {X 0.185,Y -693.434,Z 596.444,A 0.000,B 0.000,C 90.000,E1 295.976} C_DIS
LIN {X -0.191,Y -693.320,Z 596.443,A 0.000,B 0.000,C 90.000,E1 295.771} C_DIS
LIN {X -0.244,Y -693.075,Z 596.442,A 0.000,B 0.000,C 90.000,E1 295.540} C_DIS
LIN {X 0.003,Y -692.599,Z 596.440,A 0.000,B 0.000,C 90.000,E1 295.283} C_DIS
LIN {X -0.017,Y -689.725,Z 596.437,A 0.000,B 0.000,C 90.000,E1 294.695} C_DIS
LIN {X -0.185,Y -688.776,Z 596.437,A 0.000,B 0.000,C 90.000,E1 294.591} C_DIS
LIN {X -0.068,Y -687.319,Z 596.436,A 0.000,B 0.000,C 90.000,E1 294.463} C_DIS
LIN {X 0.049,Y -685.305,Z 596.435,A 0.000,B 0.000,C 90.000,E1 294.335} C_DIS
LIN {X -0.040,Y -681.371,Z 596.434,A 0.000,B 0.000,C 90.000,E1 294.079} C_DIS
LIN {X 0.336,Y -679.229,Z 596.433,A 0.000,B 0.000,C 90.000,E1 293.951} C_DIS
LIN {X 0.159,Y -670.988,Z 596.432,A 0.000,B 0.000,C 90.000,E1 293.718} C_DIS
LIN {X -0.170,Y -669.103,Z 596.432,A 0.000,B 0.000,C 90.000,E1 293.695} C_DIS
LIN {X 0.204,Y -660.663,Z 596.431,A 0.000,B 0.000,C 90.000,E1 293.515} C_DIS
LIN {X 0.194,Y -647.477,Z 596.430,A 0.000,B 0.000,C 90.000,E1 293.334} C_DIS
LIN {X -0.280,Y -637.868,Z 596.429,A 0.000,B 0.000,C 90.000,E1 293.206} C_DIS
LIN {X 0.202,Y -628.175,Z 596.428,A 0.000,B 0.000,C 90.000,E1 292.950} C_DIS
LIN {X -0.163,Y -621.808,Z 596.427,A 0.000,B 0.000,C 90.000,E1 292.823} C_DIS
LIN {X -0.217,Y -604.901,Z 596.424,A 0.000,B 0.000,C 90.000,E1 292.333} C_DIS
LIN {X 0.248,Y -578.834,Z 596.419,A 0.000,B 0.000,C 90.000,E1 291.461} C_DIS
LIN {X 0.103,Y -566.884,Z 596.417,A 0.000,B 0.000,C 90.000,E1 291.099} C_DIS
LIN {X 0.059,Y -565.358,Z 596.417,A 0.000,B 0.000,C 90.000,E1 291.046} C_DIS
LIN {X 0.226,Y -560.960,Z 596.416,A 0.000,B 0.000,C 90.000,E1 290.791} C_DIS
LIN {X 0.171,Y -560.915,Z 596.416,A 0.000,B 0.000,C 90.000,E1 290.791} C_DIS
LIN {X 0.198,Y -559.726,Z 596.415,A 0.000,B 0.000,C 90.000,E1 290.610} C_DIS
LIN {X 0.156,Y -559.718,Z 596.415,A 0.000,B 0.000,C 90.000,E1 290.610} C_DIS
LIN {X -0.194,Y -559.114,Z 596.412,A 0.000,B 0.000,C 90.000,E1 290.248} C_DIS
LIN {X 0.081,Y -558.972,Z 596.402,A 0.000,B 0.000,C 90.000,E1 288.417} C_DIS
LIN {X -0.139,Y -558.723,Z 596.396,A 0.000,B 0.000,C 90.000,E1 287.330} C_DIS
LIN {X 0.296,Y -558.256,Z 596.389,A 0.000,B 0.000,C 90.000,E1 285.898} C_DIS
LIN {X -0.097,Y -557.750,Z 596.382,A 0.000,B 0.000,C 90.000,E1 284.828} C_DIS
LIN {X -0.233,Y -556.923,Z 596.373,A 0.000,B 0.000,C 90.000,E1 283.175} C_DIS
LIN {X 0.168,Y -555.800,Z 596.362,A 0.000,B 0.000,C 90.000,E1 281.186} C_DIS
LIN {X -0.108,Y -554.729,Z 596.351,A 0.000,B 0.000,C 90.000,E1 279.265} C_DIS
LIN {X 0.048,Y -553.761,Z 596.341,A 0.000,B 0.000,C 90.000,E1 277.296} C_DIS
LIN {X 0.103,Y -552.873,Z 596.330,A 0.000,B 0.000,C 90.000,E1 275.334} C_DIS
LIN {X 0.042,Y -552.167,Z 596.319,A 0.000,B 0.000,C 90.000,E1 273.383} C_DIS
LIN {X -0.035,Y -551.653,Z 596.308,A 0.000,B 0.000,C 90.000,E1 271.432} C_DIS
LIN {X 0.271,Y -551.326,Z 596.300,A 0.000,B 0.000,C 90.000,E1 270.000} C_DIS
LIN {X 0.078,Y -550.714,Z 596.291,A 0.000,B 0.000,C 90.000,E1 268.339} C_DIS
LIN {X -0.092,Y -550.060,Z 596.281,A 0.000,B 0.000,C 90.000,E1 266.674} C_DIS
LIN {X 0.192,Y -549.394,Z 596.274,A 0.000,B 0.000,C 90.000,E1 265.241} C_DIS
LIN {X 0.005,Y -548.610,Z 596.266,A 0.000,B 0.000,C 90.000,E1 263.856} C_DIS
LIN {X 0.262,Y -547.808,Z 596.260,A 0.000,B 0.000,C 90.000,E1 262.704} C_DIS
LIN {X 0.142,Y -546.319,Z 596.250,A 0.000,B 0.000,C 90.000,E1 261.027} C_DIS
LIN {X 0.163,Y -544.399,Z 596.239,A 0.000,B 0.000,C 90.000,E1 259.050} C_DIS
LIN {X 0.069,Y -543.069,Z 596.231,A 0.000,B 0.000,C 90.000,E1 257.645} C_DIS
LIN {X 0.152,Y -541.315,Z 596.222,A 0.000,B 0.000,C 90.000,E1 255.936} C_DIS
LIN {X -0.013,Y -540.474,Z 596.217,A 0.000,B 0.000,C 90.000,E1 255.102} C_DIS
LIN {X 0.155,Y -538.746,Z 596.208,A 0.000,B 0.000,C 90.000,E1 253.378} C_DIS
LIN {X 0.221,Y -537.220,Z 596.200,A 0.000,B 0.000,C 90.000,E1 251.945} C_DIS
LIN {X 0.174,Y -536.305,Z 596.195,A 0.000,B 0.000,C 90.000,E1 251.094} C_DIS
LIN {X -0.150,Y -534.347,Z 596.187,A 0.000,B 0.000,C 90.000,E1 249.699} C_DIS
LIN {X -0.028,Y -532.415,Z 596.181,A 0.000,B 0.000,C 90.000,E1 248.539} C_DIS
LIN {X -0.039,Y -529.756,Z 596.173,A 0.000,B 0.000,C 90.000,E1 247.102} C_DIS
LIN {X -0.092,Y -526.918,Z 596.165,A 0.000,B 0.000,C 90.000,E1 245.665} C_DIS
LIN {X 0.022,Y -523.926,Z 596.157,A 0.000,B 0.000,C 90.000,E1 244.204} C_DIS
LIN {X -0.066,Y -521.397,Z 596.150,A 0.000,B 0.000,C 90.000,E1 243.050} C_DIS
LIN {X -0.067,Y -518.053,Z 596.142,A 0.000,B 0.000,C 90.000,E1 241.591} C_DIS
LIN {X -0.009,Y -515.152,Z 596.136,A 0.000,B 0.000,C 90.000,E1 240.411} C_DIS
LIN {X -0.207,Y -509.242,Z 596.123,A 0.000,B 0.000,C 90.000,E1 238.074} C_DIS
LIN {X 0.251,Y -506.238,Z 596.116,A 0.000,B 0.000,C 90.000,E1 236.834} C_DIS
LIN {X -0.036,Y -502.858,Z 596.109,A 0.000,B 0.000,C 90.000,E1 235.674} C_DIS
LIN {X -0.089,Y -499.376,Z 596.103,A 0.000,B 0.000,C 90.000,E1 234.482} C_DIS
LIN {X 0.101,Y -492.112,Z 596.088,A 0.000,B 0.000,C 90.000,E1 231.743} C_DIS
LIN {X 0.164,Y -487.325,Z 596.077,A 0.000,B 0.000,C 90.000,E1 229.908} C_DIS
LIN {X 0.105,Y -484.119,Z 596.071,A 0.000,B 0.000,C 90.000,E1 228.690} C_DIS
LIN {X -0.076,Y -479.525,Z 596.060,A 0.000,B 0.000,C 90.000,E1 226.863} C_DIS
LIN {X -0.054,Y -475.015,Z 596.050,A 0.000,B 0.000,C 90.000,E1 225.000} C_DIS
LIN {X -0.224,Y -471.405,Z 596.041,A 0.000,B 0.000,C 90.000,E1 223.461} C_DIS
LIN {X -0.019,Y -467.029,Z 596.031,A 0.000,B 0.000,C 90.000,E1 221.553} C_DIS
LIN {X 0.039,Y -463.584,Z 596.022,A 0.000,B 0.000,C 90.000,E1 219.967} C_DIS
LIN {X -0.233,Y -459.588,Z 596.012,A 0.000,B 0.000,C 90.000,E1 218.096} C_DIS
LIN {X 0.008,Y -456.952,Z 596.004,A 0.000,B 0.000,C 90.000,E1 216.790} C_DIS
LIN {X 0.029,Y -453.802,Z 595.996,A 0.000,B 0.000,C 90.000,E1 215.185} C_DIS
LIN {X -0.131,Y -448.873,Z 595.981,A 0.000,B 0.000,C 90.000,E1 212.625} C_DIS
LIN {X -0.064,Y -445.392,Z 595.970,A 0.000,B 0.000,C 90.000,E1 210.669} C_DIS
LIN {X 0.184,Y -443.042,Z 595.963,A 0.000,B 0.000,C 90.000,E1 209.333} C_DIS
LIN {X 0.085,Y -438.967,Z 595.950,A 0.000,B 0.000,C 90.000,E1 207.052} C_DIS
LIN {X 0.030,Y -436.081,Z 595.941,A 0.000,B 0.000,C 90.000,E1 205.412} C_DIS
LIN {X -0.077,Y -432.690,Z 595.930,A 0.000,B 0.000,C 90.000,E1 203.439} C_DIS
LIN {X 0.181,Y -429.411,Z 595.919,A 0.000,B 0.000,C 90.000,E1 201.408} C_DIS
LIN {X 0.014,Y -425.734,Z 595.906,A 0.000,B 0.000,C 90.000,E1 199.087} C_DIS
LIN {X -0.177,Y -422.821,Z 595.895,A 0.000,B 0.000,C 90.000,E1 197.094} C_DIS
LIN {X -0.103,Y -419.606,Z 595.882,A 0.000,B 0.000,C 90.000,E1 194.717} C_DIS
LIN {X -0.074,Y -417.691,Z 595.874,A 0.000,B 0.000,C 90.000,E1 193.355} C_DIS
LIN {X 0.056,Y -414.190,Z 595.861,A 0.000,B 0.000,C 90.000,E1 190.950} C_DIS
LIN {X -0.007,Y -410.195,Z 595.844,A 0.000,B 0.000,C 90.000,E1 187.871} C_DIS
LIN {X 0.039,Y -408.523,Z 595.836,A 0.000,B 0.000,C 90.000,E1 186.486} C_DIS
LIN {X -0.034,Y -405.029,Z 595.821,A 0.000,B 0.000,C 90.000,E1 183.726} C_DIS
LIN {X 0.032,Y -401.423,Z 595.799,A 0.000,B 0.000,C 90.000,E1 179.885} C_DIS
LIN {X 0.058,Y -399.313,Z 595.782,A 0.000,B 0.000,C 90.000,E1 176.731} C_DIS
LIN {X 0.126,Y -398.131,Z 595.766,A 0.000,B 0.000,C 90.000,E1 173.913} C_DIS
LIN {X -0.110,Y -397.623,Z 595.755,A 0.000,B 0.000,C 90.000,E1 171.837} C_DIS
LIN {X 0.092,Y -397.356,Z 595.739,A 0.000,B 0.000,C 90.000,E1 168.993} C_DIS
LIN {X 0.069,Y -397.540,Z 595.725,A 0.000,B 0.000,C 90.000,E1 166.533} C_DIS
LIN {X -0.111,Y -397.972,Z 595.714,A 0.000,B 0.000,C 90.000,E1 164.448} C_DIS
LIN {X -0.195,Y -398.726,Z 595.700,A 0.000,B 0.000,C 90.000,E1 162.000} C_DIS
LIN {X -0.021,Y -399.548,Z 595.686,A 0.000,B 0.000,C 90.000,E1 159.518} C_DIS
LIN {X 0.079,Y -400.544,Z 595.673,A 0.000,B 0.000,C 90.000,E1 157.050} C_DIS
LIN {X -0.082,Y -401.466,Z 595.661,A 0.000,B 0.000,C 90.000,E1 154.973} C_DIS
LIN {X -0.047,Y -402.430,Z 595.649,A 0.000,B 0.000,C 90.000,E1 152.871} C_DIS
LIN {X 0.042,Y -403.018,Z 595.642,A 0.000,B 0.000,C 90.000,E1 151.463} C_DIS
LIN {X -0.126,Y -403.736,Z 595.632,A 0.000,B 0.000,C 90.000,E1 149.744} C_DIS
LIN {X -0.070,Y -404.332,Z 595.622,A 0.000,B 0.000,C 90.000,E1 147.995} C_DIS
LIN {X 0.217,Y -404.749,Z 595.613,A 0.000,B 0.000,C 90.000,E1 146.215} C_DIS
LIN {X 0.176,Y -405.182,Z 595.603,A 0.000,B 0.000,C 90.000,E1 144.482} C_DIS
LIN {X -0.059,Y -405.697,Z 595.591,A 0.000,B 0.000,C 90.000,E1 142.431} C_DIS
LIN {X -0.108,Y -406.288,Z 595.580,A 0.000,B 0.000,C 90.000,E1 140.356} C_DIS
LIN {X 0.124,Y -406.825,Z 595.568,A 0.000,B 0.000,C 90.000,E1 138.243} C_DIS
LIN {X 0.079,Y -407.024,Z 595.560,A 0.000,B 0.000,C 90.000,E1 136.863} C_DIS
LIN {X -0.009,Y -407.361,Z 595.549,A 0.000,B 0.000,C 90.000,E1 134.798} C_DIS
LIN {X 0.209,Y -407.611,Z 595.537,A 0.000,B 0.000,C 90.000,E1 132.690} C_DIS
LIN {X 0.164,Y -407.786,Z 595.526,A 0.000,B 0.000,C 90.000,E1 130.620} C_DIS
LIN {X 0.021,Y -407.911,Z 595.516,A 0.000,B 0.000,C 90.000,E1 128.910} C_DIS
LIN {X -0.095,Y -407.918,Z 595.515,A 0.000,B 0.000,C 90.000,E1 128.624} C_DIS
LIN {X 0.146,Y -415.101,Z 595.501,A 0.000,B 0.000,C 90.000,E1 126.091} C_DIS
LIN {X -0.260,Y -416.021,Z 595.499,A 0.000,B 0.000,C 90.000,E1 125.804} C_DIS
LIN {X 0.206,Y -425.530,Z 595.478,A 0.000,B 0.000,C 90.000,E1 122.005} C_DIS
LIN {X 0.148,Y -426.516,Z 595.476,A 0.000,B 0.000,C 90.000,E1 121.671} C_DIS
LIN {X 0.109,Y -426.545,Z 595.476,A 0.000,B 0.000,C 90.000,E1 121.671} C_DIS
LIN {X -0.093,Y -436.815,Z 595.473,A 0.000,B 0.000,C 90.000,E1 121.209} C_DIS
LIN {X -0.045,Y -440.281,Z 595.473,A 0.000,B 0.000,C 90.000,E1 121.052} C_DIS
LIN {X 0.038,Y -446.763,Z 595.471,A 0.000,B 0.000,C 90.000,E1 120.718} C_DIS
LIN {X 0.002,Y -453.450,Z 595.469,A 0.000,B 0.000,C 90.000,E1 120.413} C_DIS
LIN {X -0.050,Y -466.880,Z 595.465,A 0.000,B 0.000,C 90.000,E1 119.745} C_DIS
LIN {X -0.174,Y -473.517,Z 595.463,A 0.000,B 0.000,C 90.000,E1 119.411} C_DIS
LIN {X -0.040,Y -480.291,Z 595.461,A 0.000,B 0.000,C 90.000,E1 119.027} C_DIS
LIN {X 0.294,Y -486.743,Z 595.459,A 0.000,B 0.000,C 90.000,E1 118.615} C_DIS
LIN {X 0.097,Y -494.777,Z 595.457,A 0.000,B 0.000,C 90.000,E1 118.153} C_DIS
LIN {X 0.279,Y -502.567,Z 595.454,A 0.000,B 0.000,C 90.000,E1 117.641} C_DIS
LIN {X 0.072,Y -508.737,Z 595.452,A 0.000,B 0.000,C 90.000,E1 117.257} C_DIS
LIN {X 0.032,Y -511.649,Z 595.450,A 0.000,B 0.000,C 90.000,E1 117.052} C_DIS
LIN {X 0.208,Y -515.858,Z 595.449,A 0.000,B 0.000,C 90.000,E1 116.744} C_DIS
LIN {X 0.005,Y -523.205,Z 595.446,A 0.000,B 0.000,C 90.000,E1 116.232} C_DIS
LIN {X -0.062,Y -530.589,Z 595.443,A 0.000,B 0.000,C 90.000,E1 115.668} C_DIS
LIN {X -0.110,Y -536.422,Z 595.440,A 0.000,B 0.000,C 90.000,E1 115.207} C_DIS
LIN {X -0.062,Y -540.698,Z 595.438,A 0.000,B 0.000,C 90.000,E1 114.847} C_DIS
LIN {X 0.048,Y -545.759,Z 595.436,A 0.000,B 0.000,C 90.000,E1 114.387} C_DIS
LIN {X 0.168,Y -550.868,Z 595.433,A 0.000,B 0.000,C 90.000,E1 113.898} C_DIS
LIN {X -0.231,Y -556.400,Z 595.430,A 0.000,B 0.000,C 90.000,E1 113.334} C_DIS
LIN {X -0.033,Y -560.582,Z 595.427,A 0.000,B 0.000,C 90.000,E1 112.823} C_DIS
LIN {X -0.248,Y -565.603,Z 595.423,A 0.000,B 0.000,C 90.000,E1 112.153} C_DIS
LIN {X -0.205,Y -569.905,Z 595.419,A 0.000,B 0.000,C 90.000,E1 111.461} C_DIS
LIN {X 0.114,Y -574.373,Z 595.415,A 0.000,B 0.000,C 90.000,E1 110.610} C_DIS
LIN {X -0.056,Y -578.449,Z 595.410,A 0.000,B 0.000,C 90.000,E1 109.812} C_DIS
LIN {X -0.111,Y -581.561,Z 595.406,A 0.000,B 0.000,C 90.000,E1 109.141} C_DIS
LIN {X -0.066,Y -583.951,Z 595.403,A 0.000,B 0.000,C 90.000,E1 108.598} C_DIS
LIN {X 0.223,Y -587.219,Z 595.399,A 0.000,B 0.000,C 90.000,E1 107.764} C_DIS
LIN {X -0.156,Y -591.013,Z 595.393,A 0.000,B 0.000,C 90.000,E1 106.732} C_DIS
LIN {X -0.215,Y -592.809,Z 595.390,A 0.000,B 0.000,C 90.000,E1 106.205} C_DIS
LIN {X -0.121,Y -596.247,Z 595.384,A 0.000,B 0.000,C 90.000,E1 105.134} C_DIS
LIN {X -0.249,Y -602.136,Z 595.374,A 0.000,B 0.000,C 90.000,E1 103.300} C_DIS
LIN {X 0.151,Y -606.338,Z 595.367,A 0.000,B 0.000,C 90.000,E1 101.951} C_DIS
LIN {X 0.027,Y -610.727,Z 595.359,A 0.000,B 0.000,C 90.000,E1 100.658} C_DIS
LIN {X 0.103,Y -614.048,Z 595.354,A 0.000,B 0.000,C 90.000,E1 99.613} C_DIS
LIN {X 0.226,Y -617.210,Z 595.348,A 0.000,B 0.000,C 90.000,E1 98.568} C_DIS
LIN {X 0.065,Y -621.031,Z 595.341,A 0.000,B 0.000,C 90.000,E1 97.296} C_DIS
LIN {X 0.199,Y -623.919,Z 595.335,A 0.000,B 0.000,C 90.000,E1 96.258} C_DIS
LIN {X -0.015,Y -625.902,Z 595.331,A 0.000,B 0.000,C 90.000,E1 95.511} C_DIS
LIN {X -0.155,Y -627.760,Z 595.326,A 0.000,B 0.000,C 90.000,E1 94.759} C_DIS
LIN {X 0.291,Y -629.322,Z 595.322,A 0.000,B 0.000,C 90.000,E1 93.955} C_DIS
LIN {X -0.148,Y -631.257,Z 595.317,A 0.000,B 0.000,C 90.000,E1 92.980} C_DIS
LIN {X -0.200,Y -633.183,Z 595.310,A 0.000,B 0.000,C 90.000,E1 91.718} C_DIS
LIN {X 0.282,Y -634.200,Z 595.305,A 0.000,B 0.000,C 90.000,E1 90.917} C_DIS
LIN {X 0.144,Y -634.997,Z 595.301,A 0.000,B 0.000,C 90.000,E1 90.172} C_DIS
LIN {X 0.014,Y -635.532,Z 595.297,A 0.000,B 0.000,C 90.000,E1 89.427} C_DIS
LIN {X -0.113,Y -635.827,Z 595.293,A 0.000,B 0.000,C 90.000,E1 88.682} C_DIS
LIN {X -0.219,Y -635.901,Z 595.288,A 0.000,B 0.000,C 90.000,E1 87.936} C_DIS
LIN {X -0.188,Y -635.573,Z 595.281,A 0.000,B 0.000,C 90.000,E1 86.674} C_DIS
LIN {X -0.286,Y -635.108,Z 595.277,A 0.000,B 0.000,C 90.000,E1 85.927} C_DIS
LIN {X -0.017,Y -634.270,Z 595.272,A 0.000,B 0.000,C 90.000,E1 84.894} C_DIS
LIN {X 0.019,Y -632.892,Z 595.265,A 0.000,B 0.000,C 90.000,E1 83.628} C_DIS
LIN {X 0.163,Y -632.228,Z 595.262,A 0.000,B 0.000,C 90.000,E1 83.109} C_DIS
LIN {X -0.188,Y -630.555,Z 595.256,A 0.000,B 0.000,C 90.000,E1 82.129} C_DIS
LIN {X -0.267,Y -629.130,Z 595.252,A 0.000,B 0.000,C 90.000,E1 81.376} C_DIS
LIN {X 0.053,Y -627.001,Z 595.246,A 0.000,B 0.000,C 90.000,E1 80.330} C_DIS
LIN {X -0.273,Y -624.720,Z 595.241,A 0.000,B 0.000,C 90.000,E1 79.342} C_DIS
LIN {X -0.112,Y -621.559,Z 595.234,A 0.000,B 0.000,C 90.000,E1 78.049} C_DIS
LIN {X -0.157,Y -619.548,Z 595.229,A 0.000,B 0.000,C 90.000,E1 77.285} C_DIS
LIN {X -0.076,Y -615.838,Z 595.222,A 0.000,B 0.000,C 90.000,E1 75.992} C_DIS
LIN {X 0.169,Y -612.652,Z 595.216,A 0.000,B 0.000,C 90.000,E1 74.936} C_DIS
LIN {X 0.186,Y -610.116,Z 595.212,A 0.000,B 0.000,C 90.000,E1 74.157} C_DIS
LIN {X 0.181,Y -607.304,Z 595.208,A 0.000,B 0.000,C 90.000,E1 73.378} C_DIS
LIN {X 0.149,Y -604.195,Z 595.203,A 0.000,B 0.000,C 90.000,E1 72.598} C_DIS
LIN {X 0.085,Y -600.861,Z 595.199,A 0.000,B 0.000,C 90.000,E1 71.819} C_DIS
LIN {X -0.068,Y -596.570,Z 595.194,A 0.000,B 0.000,C 90.000,E1 70.913} C_DIS
LIN {X -0.279,Y -591.925,Z 595.189,A 0.000,B 0.000,C 90.000,E1 70.007} C_DIS
LIN {X -0.182,Y -587.630,Z 595.184,A 0.000,B 0.000,C 90.000,E1 69.209} C_DIS
LIN {X -0.229,Y -582.817,Z 595.180,A 0.000,B 0.000,C 90.000,E1 68.411} C_DIS
LIN {X -0.035,Y -578.458,Z 595.176,A 0.000,B 0.000,C 90.000,E1 67.720} C_DIS
LIN {X -0.099,Y -573.586,Z 595.172,A 0.000,B 0.000,C 90.000,E1 67.050} C_DIS
LIN {X 0.100,Y -569.348,Z 595.169,A 0.000,B 0.000,C 90.000,E1 66.485} C_DIS
LIN {X 0.267,Y -564.692,Z 595.166,A 0.000,B 0.000,C 90.000,E1 65.921} C_DIS
LIN {X -0.061,Y -559.686,Z 595.163,A 0.000,B 0.000,C 90.000,E1 65.409} C_DIS
LIN {X -0.133,Y -554.777,Z 595.161,A 0.000,B 0.000,C 90.000,E1 64.921} C_DIS
LIN {X 0.169,Y -549.441,Z 595.158,A 0.000,B 0.000,C 90.000,E1 64.409} C_DIS
LIN {X -0.001,Y -543.729,Z 595.155,A 0.000,B 0.000,C 90.000,E1 63.973} C_DIS
LIN {X -0.104,Y -537.692,Z 595.153,A 0.000,B 0.000,C 90.000,E1 63.563} C_DIS
LIN {X -0.131,Y -532.624,Z 595.151,A 0.000,B 0.000,C 90.000,E1 63.256} C_DIS
LIN {X 0.064,Y -527.591,Z 595.150,A 0.000,B 0.000,C 90.000,E1 62.948} C_DIS
LIN {X -0.175,Y -519.041,Z 595.147,A 0.000,B 0.000,C 90.000,E1 62.538} C_DIS
LIN {X -0.114,Y -513.736,Z 595.146,A 0.000,B 0.000,C 90.000,E1 62.281} C_DIS
LIN {X 0.074,Y -501.768,Z 595.143,A 0.000,B 0.000,C 90.000,E1 61.719} C_DIS
LIN {X 0.151,Y -479.478,Z 595.137,A 0.000,B 0.000,C 90.000,E1 60.717} C_DIS
LIN {X 0.058,Y -462.617,Z 595.133,A 0.000,B 0.000,C 90.000,E1 59.950} C_DIS
LIN {X 0.029,Y -449.428,Z 595.129,A 0.000,B 0.000,C 90.000,E1 59.282} C_DIS
LIN {X -0.015,Y -449.324,Z 595.129,A 0.000,B 0.000,C 90.000,E1 59.282} C_DIS
LIN {X -0.286,Y -444.256,Z 595.115,A 0.000,B 0.000,C 90.000,E1 56.707} C_DIS
LIN {X 0.018,Y -443.578,Z 595.113,A 0.000,B 0.000,C 90.000,E1 56.342} C_DIS
LIN {X 0.030,Y -434.485,Z 595.091,A 0.000,B 0.000,C 90.000,E1 52.396} C_DIS
LIN {X -0.044,Y -432.609,Z 595.086,A 0.000,B 0.000,C 90.000,E1 51.412} C_DIS
LIN {X -0.031,Y -434.255,Z 595.074,A 0.000,B 0.000,C 90.000,E1 49.337} C_DIS
LIN {X -0.008,Y -435.545,Z 595.065,A 0.000,B 0.000,C 90.000,E1 47.676} C_DIS
LIN {X 0.020,Y -437.120,Z 595.054,A 0.000,B 0.000,C 90.000,E1 45.688} C_DIS
LIN {X 0.060,Y -438.661,Z 595.043,A 0.000,B 0.000,C 90.000,E1 43.704} C_DIS
LIN {X 0.216,Y -439.500,Z 595.036,A 0.000,B 0.000,C 90.000,E1 42.366} C_DIS
LIN {X 0.090,Y -440.219,Z 595.028,A 0.000,B 0.000,C 90.000,E1 41.067} C_DIS
LIN {X -0.014,Y -440.892,Z 595.019,A 0.000,B 0.000,C 90.000,E1 39.439} C_DIS
LIN {X -0.102,Y -441.550,Z 595.010,A 0.000,B 0.000,C 90.000,E1 37.810} C_DIS
LIN {X -0.102,Y -441.940,Z 595.001,A 0.000,B 0.000,C 90.000,E1 36.171} C_DIS
LIN {X 0.219,Y -442.179,Z 594.994,A 0.000,B 0.000,C 90.000,E1 34.818} C_DIS
LIN {X 0.289,Y -442.252,Z 594.986,A 0.000,B 0.000,C 90.000,E1 33.499} C_DIS
LIN {X -0.159,Y -442.405,Z 594.975,A 0.000,B 0.000,C 90.000,E1 31.592} C_DIS
LIN {X 0.045,Y -442.472,Z 594.968,A 0.000,B 0.000,C 90.000,E1 30.256} C_DIS
LIN {X -0.079,Y -442.613,Z 594.957,A 0.000,B 0.000,C 90.000,E1 28.309} C_DIS
LIN {X -0.196,Y -442.845,Z 594.946,A 0.000,B 0.000,C 90.000,E1 26.360} C_DIS
LIN {X 0.141,Y -443.189,Z 594.934,A 0.000,B 0.000,C 90.000,E1 24.027} C_DIS
LIN {X 0.038,Y -443.536,Z 594.923,A 0.000,B 0.000,C 90.000,E1 22.078} C_DIS
LIN {X 0.016,Y -443.959,Z 594.912,A 0.000,B 0.000,C 90.000,E1 20.120} C_DIS
LIN {X 0.136,Y -444.566,Z 594.899,A 0.000,B 0.000,C 90.000,E1 17.819} C_DIS
LIN {X 0.009,Y -445.323,Z 594.886,A 0.000,B 0.000,C 90.000,E1 15.552} C_DIS
LIN {X 0.063,Y -446.478,Z 594.872,A 0.000,B 0.000,C 90.000,E1 12.939} C_DIS
LIN {X -0.161,Y -447.994,Z 594.858,A 0.000,B 0.000,C 90.000,E1 10.366} C_DIS
LIN {X 0.012,Y -449.273,Z 594.847,A 0.000,B 0.000,C 90.000,E1 8.398} C_DIS
LIN {X -0.086,Y -451.054,Z 594.834,A 0.000,B 0.000,C 90.000,E1 6.144} C_DIS
LIN {X -0.028,Y -453.405,Z 594.820,A 0.000,B 0.000,C 90.000,E1 3.555} C_DIS
LIN {X 0.042,Y -456.131,Z 594.805,A 0.000,B 0.000,C 90.000,E1 0.974} C_DIS
LIN {X -0.171,Y -458.790,Z 594.794,A 0.000,B 0.000,C 90.000,E1 358.854} C_DIS
LIN {X -0.186,Y -462.843,Z 594.778,A 0.000,B 0.000,C 90.000,E1 355.988} C_DIS
LIN {X -0.221,Y -465.728,Z 594.767,A 0.000,B 0.000,C 90.000,E1 354.090} C_DIS
LIN {X -0.139,Y -468.689,Z 594.757,A 0.000,B 0.000,C 90.000,E1 352.186} C_DIS
LIN {X 0.076,Y -471.609,Z 594.746,A 0.000,B 0.000,C 90.000,E1 350.274} C_DIS
LIN {X -0.096,Y -475.062,Z 594.734,A 0.000,B 0.000,C 90.000,E1 348.105} C_DIS
LIN {X 0.030,Y -477.737,Z 594.725,A 0.000,B 0.000,C 90.000,E1 346.533} C_DIS
LIN {X 0.098,Y -482.198,Z 594.711,A 0.000,B 0.000,C 90.000,E1 344.047} C_DIS
LIN {X -0.073,Y -484.517,Z 594.705,A 0.000,B 0.000,C 90.000,E1 342.834} C_DIS
LIN {X 0.020,Y -489.200,Z 594.691,A 0.000,B 0.000,C 90.000,E1 340.369} C_DIS
LIN {X -0.007,Y -492.153,Z 594.683,A 0.000,B 0.000,C 90.000,E1 338.847} C_DIS
LIN {X -0.261,Y -494.862,Z 594.674,A 0.000,B 0.000,C 90.000,E1 337.358} C_DIS
LIN {X 0.190,Y -497.483,Z 594.666,A 0.000,B 0.000,C 90.000,E1 335.793} C_DIS
LIN {X 0.177,Y -499.402,Z 594.659,A 0.000,B 0.000,C 90.000,E1 334.588} C_DIS
LIN {X -0.192,Y -501.760,Z 594.651,A 0.000,B 0.000,C 90.000,E1 333.127} C_DIS
LIN {X -0.057,Y -505.430,Z 594.637,A 0.000,B 0.000,C 90.000,E1 330.717} C_DIS
LIN {X 0.101,Y -508.604,Z 594.626,A 0.000,B 0.000,C 90.000,E1 328.614} C_DIS
LIN {X 0.009,Y -512.054,Z 594.614,A 0.000,B 0.000,C 90.000,E1 326.548} C_DIS
LIN {X 0.162,Y -514.699,Z 594.606,A 0.000,B 0.000,C 90.000,E1 325.055} C_DIS
LIN {X -0.190,Y -517.491,Z 594.598,A 0.000,B 0.000,C 90.000,E1 323.623} C_DIS
LIN {X 0.039,Y -519.221,Z 594.593,A 0.000,B 0.000,C 90.000,E1 322.718} C_DIS
LIN {X -0.257,Y -525.950,Z 594.575,A 0.000,B 0.000,C 90.000,E1 319.542} C_DIS
LIN {X -0.028,Y -528.606,Z 594.570,A 0.000,B 0.000,C 90.000,E1 318.647} C_DIS
LIN {X 0.159,Y -530.764,Z 594.568,A 0.000,B 0.000,C 90.000,E1 318.162} C_DIS
LIN {X -0.057,Y -531.892,Z 594.567,A 0.000,B 0.000,C 90.000,E1 318.038} C_DIS
LIN {X -0.120,Y -533.592,Z 594.565,A 0.000,B 0.000,C 90.000,E1 317.757} C_DIS
LIN {X -0.140,Y -536.024,Z 594.564,A 0.000,B 0.000,C 90.000,E1 317.472} C_DIS
LIN {X 0.036,Y -537.050,Z 594.563,A 0.000,B 0.000,C 90.000,E1 317.310} C_DIS
LIN {X 0.117,Y -541.274,Z 594.560,A 0.000,B 0.000,C 90.000,E1 316.863} C_DIS
LIN {X -0.270,Y -546.206,Z 594.558,A 0.000,B 0.000,C 90.000,E1 316.458} C_DIS
LIN {X 0.054,Y -555.108,Z 594.554,A 0.000,B 0.000,C 90.000,E1 315.729} C_DIS
LIN {X 0.091,Y -566.982,Z 594.549,A 0.000,B 0.000,C 90.000,E1 314.838} C_DIS
LIN {X 0.036,Y -572.904,Z 594.547,A 0.000,B 0.000,C 90.000,E1 314.393} C_DIS
LIN {X 0.004,Y -581.810,Z 594.543,A 0.000,B 0.000,C 90.000,E1 313.743} C_DIS
LIN {X 0.091,Y -590.577,Z 594.539,A 0.000,B 0.000,C 90.000,E1 313.095} C_DIS
LIN {X -0.240,Y -596.237,Z 594.537,A 0.000,B 0.000,C 90.000,E1 312.690} C_DIS
LIN {X 0.212,Y -603.126,Z 594.534,A 0.000,B 0.000,C 90.000,E1 312.081} C_DIS
LIN {X 0.315,Y -608.309,Z 594.531,A 0.000,B 0.000,C 90.000,E1 311.595} C_DIS
LIN {X -0.132,Y -613.479,Z 594.529,A 0.000,B 0.000,C 90.000,E1 311.148} C_DIS
LIN {X -0.349,Y -619.452,Z 594.525,A 0.000,B 0.000,C 90.000,E1 310.539} C_DIS
LIN {X -0.191,Y -624.140,Z 594.522,A 0.000,B 0.000,C 90.000,E1 310.011} C_DIS
LIN {X -0.185,Y -632.885,Z 594.517,A 0.000,B 0.000,C 90.000,E1 308.991} C_DIS
LIN {X -0.057,Y -641.007,Z 594.511,A 0.000,B 0.000,C 90.000,E1 307.971} C_DIS
LIN {X -0.257,Y -645.708,Z 594.508,A 0.000,B 0.000,C 90.000,E1 307.363} C_DIS
LIN {X 0.091,Y -650.065,Z 594.504,A 0.000,B 0.000,C 90.000,E1 306.710} C_DIS
LIN {X 0.060,Y -653.262,Z 594.501,A 0.000,B 0.000,C 90.000,E1 306.217} C_DIS
LIN {X 0.089,Y -656.963,Z 594.498,A 0.000,B 0.000,C 90.000,E1 305.598} C_DIS
LIN {X 0.107,Y -659.640,Z 594.495,A 0.000,B 0.000,C 90.000,E1 305.105} C_DIS
LIN {X 0.141,Y -662.133,Z 594.492,A 0.000,B 0.000,C 90.000,E1 304.612} C_DIS
LIN {X -0.246,Y -665.543,Z 594.488,A 0.000,B 0.000,C 90.000,E1 303.913} C_DIS
LIN {X -0.182,Y -667.676,Z 594.486,A 0.000,B 0.000,C 90.000,E1 303.420} C_DIS
LIN {X 0.183,Y -671.566,Z 594.480,A 0.000,B 0.000,C 90.000,E1 302.418} C_DIS
LIN {X 0.038,Y -675.284,Z 594.475,A 0.000,B 0.000,C 90.000,E1 301.465} C_DIS
LIN {X -0.070,Y -678.865,Z 594.470,A 0.000,B 0.000,C 90.000,E1 300.512} C_DIS
LIN {X 0.110,Y -682.320,Z 594.464,A 0.000,B 0.000,C 90.000,E1 299.539} C_DIS
LIN {X -0.255,Y -685.562,Z 594.459,A 0.000,B 0.000,C 90.000,E1 298.615} C_DIS
LIN {X 0.020,Y -688.578,Z 594.454,A 0.000,B 0.000,C 90.000,E1 297.641} C_DIS
LIN {X 0.097,Y -690.736,Z 594.450,A 0.000,B 0.000,C 90.000,E1 296.924} C_DIS
LIN {X -0.116,Y -692.281,Z 594.446,A 0.000,B 0.000,C 90.000,E1 296.232} C_DIS
LIN {X 0.126,Y -692.400,Z 594.444,A 0.000,B 0.000,C 90.000,E1 295.976} C_DIS
LIN {X -0.310,Y -692.153,Z 594.442,A 0.000,B 0.000,C 90.000,E1 295.540} C_DIS
LIN {X -0.065,Y -691.555,Z 594.440,A 0.000,B 0.000,C 90.000,E1 295.283} C_DIS
LIN {X -0.210,Y -689.448,Z 594.438,A 0.000,B 0.000,C 90.000,E1 294.823} C_DIS
LIN {X -0.092,Y -688.752,Z 594.437,A 0.000,B 0.000,C 90.000,E1 294.695} C_DIS
LIN {X -0.261,Y -687.680,Z 594.437,A 0.000,B 0.000,C 90.000,E1 294.591} C_DIS
LIN {X 0.113,Y -681.494,Z 594.434,A 0.000,B 0.000,C 90.000,E1 294.131} C_DIS
LIN {X -0.301,Y -680.005,Z 594.434,A 0.000,B 0.000,C 90.000,E1 294.079} C_DIS
LIN {X 0.056,Y -675.884,Z 594.433,A 0.000,B 0.000,C 90.000,E1 293.898} C_DIS
LIN {X -0.396,Y -670.247,Z 594.432,A 0.000,B 0.000,C 90.000,E1 293.770} C_DIS
LIN {X -0.049,Y -665.782,Z 594.431,A 0.000,B 0.000,C 90.000,E1 293.643} C_DIS
LIN {X 0.224,Y -659.625,Z 594.431,A 0.000,B 0.000,C 90.000,E1 293.515} C_DIS
LIN {X 0.150,Y -646.712,Z 594.430,A 0.000,B 0.000,C 90.000,E1 293.334} C_DIS
LIN {X -0.352,Y -637.225,Z 594.429,A 0.000,B 0.000,C 90.000,E1 293.206} C_DIS
LIN {X 0.106,Y -627.570,Z 594.428,A 0.000,B 0.000,C 90.000,E1 292.950} C_DIS
LIN {X 0.099,Y -617.811,Z 594.426,A 0.000,B 0.000,C 90.000,E1 292.695} C_DIS
LIN {X -0.103,Y -579.975,Z 594.420,A 0.000,B 0.000,C 90.000,E1 291.535} C_DIS
LIN {X -0.282,Y -569.412,Z 594.418,A 0.000,B 0.000,C 90.000,E1 291.227} C_DIS
LIN {X -0.129,Y -565.104,Z 594.417,A 0.000,B 0.000,C 90.000,E1 291.046} C_DIS
LIN {X 0.204,Y -561.162,Z 594.416,A 0.000,B 0.000,C 90.000,E1 290.791} C_DIS
LIN {X 0.150,Y -561.117,Z 594.416,A 0.000,B 0.000,C 90.000,E1 290.791} C_DIS
LIN {X 0.140,Y -559.965,Z 594.415,A 0.000,B 0.000,C 90.000,E1 290.610} C_DIS
LIN {X 0.156,Y -559.345,Z 594.412,A 0.000,B 0.000,C 90.000,E1 290.194} C_DIS
LIN {X 0.305,Y -559.253,Z 594.404,A 0.000,B 0.000,C 90.000,E1 288.598} C_DIS
LIN {X 0.089,Y -559.024,Z 594.397,A 0.000,B 0.000,C 90.000,E1 287.511} C_DIS
LIN {X -0.006,Y -558.569,Z 594.390,A 0.000,B 0.000,C 90.000,E1 286.134} C_DIS
LIN {X -0.260,Y -557.924,Z 594.382,A 0.000,B 0.000,C 90.000,E1 284.773} C_DIS
LIN {X 0.154,Y -557.097,Z 594.373,A 0.000,B 0.000,C 90.000,E1 283.063} C_DIS
LIN {X 0.021,Y -555.978,Z 594.362,A 0.000,B 0.000,C 90.000,E1 281.130} C_DIS
LIN {X -0.247,Y -554.909,Z 594.351,A 0.000,B 0.000,C 90.000,E1 279.208} C_DIS
LIN {X -0.205,Y -554.053,Z 594.342,A 0.000,B 0.000,C 90.000,E1 277.530} C_DIS
LIN {X -0.131,Y -553.160,Z 594.331,A 0.000,B 0.000,C 90.000,E1 275.568} C_DIS
LIN {X -0.140,Y -552.416,Z 594.320,A 0.000,B 0.000,C 90.000,E1 273.612} C_DIS
LIN {X -0.212,Y -551.897,Z 594.309,A 0.000,B 0.000,C 90.000,E1 271.661} C_DIS
LIN {X 0.098,Y -551.583,Z 594.301,A 0.000,B 0.000,C 90.000,E1 270.229} C_DIS
LIN {X -0.089,Y -551.005,Z 594.292,A 0.000,B 0.000,C 90.000,E1 268.568} C_DIS
LIN {X -0.280,Y -550.328,Z 594.283,A 0.000,B 0.000,C 90.000,E1 266.906} C_DIS
LIN {X 0.042,Y -549.691,Z 594.275,A 0.000,B 0.000,C 90.000,E1 265.469} C_DIS
LIN {X -0.192,Y -548.930,Z 594.267,A 0.000,B 0.000,C 90.000,E1 264.090} C_DIS
LIN {X 0.035,Y -548.376,Z 594.262,A 0.000,B 0.000,C 90.000,E1 263.223} C_DIS
LIN {X -0.165,Y -547.206,Z 594.255,A 0.000,B 0.000,C 90.000,E1 261.837} C_DIS
LIN {X 0.137,Y -546.209,Z 594.248,A 0.000,B 0.000,C 90.000,E1 260.679} C_DIS
LIN {X 0.153,Y -544.289,Z 594.237,A 0.000,B 0.000,C 90.000,E1 258.701} C_DIS
LIN {X 0.055,Y -542.927,Z 594.229,A 0.000,B 0.000,C 90.000,E1 257.297} C_DIS
LIN {X -0.186,Y -540.889,Z 594.219,A 0.000,B 0.000,C 90.000,E1 255.338} C_DIS
LIN {X 0.053,Y -538.880,Z 594.207,A 0.000,B 0.000,C 90.000,E1 253.323} C_DIS
LIN {X -0.182,Y -537.019,Z 594.198,A 0.000,B 0.000,C 90.000,E1 251.638} C_DIS
LIN {X 0.280,Y -535.962,Z 594.193,A 0.000,B 0.000,C 90.000,E1 250.732} C_DIS
LIN {X -0.072,Y -534.345,Z 594.187,A 0.000,B 0.000,C 90.000,E1 249.625} C_DIS
LIN {X -0.146,Y -532.945,Z 594.182,A 0.000,B 0.000,C 90.000,E1 248.773} C_DIS
LIN {X 0.144,Y -530.296,Z 594.174,A 0.000,B 0.000,C 90.000,E1 247.305} C_DIS
LIN {X -0.213,Y -526.859,Z 594.164,A 0.000,B 0.000,C 90.000,E1 245.613} C_DIS
LIN {X 0.207,Y -524.447,Z 594.158,A 0.000,B 0.000,C 90.000,E1 244.409} C_DIS
LIN {X -0.199,Y -521.320,Z 594.150,A 0.000,B 0.000,C 90.000,E1 242.999} C_DIS
LIN {X 0.040,Y -517.954,Z 594.142,A 0.000,B 0.000,C 90.000,E1 241.513} C_DIS
LIN {X 0.100,Y -515.031,Z 594.135,A 0.000,B 0.000,C 90.000,E1 240.333} C_DIS
LIN {X -0.097,Y -509.056,Z 594.122,A 0.000,B 0.000,C 90.000,E1 237.995} C_DIS
LIN {X 0.085,Y -506.027,Z 594.116,A 0.000,B 0.000,C 90.000,E1 236.786} C_DIS
LIN {X 0.074,Y -502.646,Z 594.109,A 0.000,B 0.000,C 90.000,E1 235.595} C_DIS
LIN {X -0.103,Y -498.296,Z 594.101,A 0.000,B 0.000,C 90.000,E1 234.116} C_DIS
LIN {X -0.099,Y -491.883,Z 594.087,A 0.000,B 0.000,C 90.000,E1 231.698} C_DIS
LIN {X 0.266,Y -487.073,Z 594.077,A 0.000,B 0.000,C 90.000,E1 229.828} C_DIS
LIN {X 0.154,Y -482.323,Z 594.067,A 0.000,B 0.000,C 90.000,E1 228.000} C_DIS
LIN {X 0.137,Y -478.487,Z 594.058,A 0.000,B 0.000,C 90.000,E1 226.458} C_DIS
LIN {X 0.032,Y -474.770,Z 594.050,A 0.000,B 0.000,C 90.000,E1 224.919} C_DIS
LIN {X -0.143,Y -471.179,Z 594.041,A 0.000,B 0.000,C 90.000,E1 223.380} C_DIS
LIN {X 0.056,Y -466.805,Z 594.030,A 0.000,B 0.000,C 90.000,E1 221.472} C_DIS
LIN {X -0.001,Y -464.069,Z 594.023,A 0.000,B 0.000,C 90.000,E1 220.216} C_DIS
LIN {X 0.084,Y -460.046,Z 594.013,A 0.000,B 0.000,C 90.000,E1 218.302} C_DIS
LIN {X 0.053,Y -457.404,Z 594.006,A 0.000,B 0.000,C 90.000,E1 217.030} C_DIS
LIN {X 0.077,Y -453.551,Z 593.995,A 0.000,B 0.000,C 90.000,E1 215.105} C_DIS
LIN {X -0.178,Y -449.225,Z 593.983,A 0.000,B 0.000,C 90.000,E1 212.880} C_DIS
LIN {X 0.022,Y -444.565,Z 593.968,A 0.000,B 0.000,C 90.000,E1 210.256} C_DIS
LIN {X 0.087,Y -441.604,Z 593.959,A 0.000,B 0.000,C 90.000,E1 208.615} C_DIS
LIN {X -0.082,Y -438.157,Z 593.948,A 0.000,B 0.000,C 90.000,E1 206.668} C_DIS
LIN {X 0.255,Y -434.699,Z 593.937,A 0.000,B 0.000,C 90.000,E1 204.643} C_DIS
LIN {X -0.067,Y -431.344,Z 593.926,A 0.000,B 0.000,C 90.000,E1 202.695} C_DIS
LIN {X -0.201,Y -428.693,Z 593.917,A 0.000,B 0.000,C 90.000,E1 201.046} C_DIS
LIN {X -0.186,Y -424.576,Z 593.902,A 0.000,B 0.000,C 90.000,E1 198.362} C_DIS
LIN {X 0.056,Y -421.249,Z 593.889,A 0.000,B 0.000,C 90.000,E1 195.969} C_DIS
LIN {X -0.126,Y -419.007,Z 593.879,A 0.000,B 0.000,C 90.000,E1 194.300} C_DIS
LIN {X -0.110,Y -417.057,Z 593.872,A 0.000,B 0.000,C 90.000,E1 192.939} C_DIS
LIN {X -0.083,Y -413.581,Z 593.859,A 0.000,B 0.000,C 90.000,E1 190.546} C_DIS
LIN {X -0.191,Y -410.120,Z 593.843,A 0.000,B 0.000,C 90.000,E1 187.814} C_DIS
LIN {X -0.145,Y -408.464,Z 593.836,A 0.000,B 0.000,C 90.000,E1 186.429} C_DIS
LIN {X 0.151,Y -404.221,Z 593.816,A 0.000,B 0.000,C 90.000,E1 182.922} C_DIS
LIN {X -0.149,Y -401.437,Z 593.799,A 0.000,B 0.000,C 90.000,E1 179.828} C_DIS
LIN {X -0.119,Y -399.354,Z 593.781,A 0.000,B 0.000,C 90.000,E1 176.674} C_DIS
LIN {X 0.035,Y -398.428,Z 593.770,A 0.000,B 0.000,C 90.000,E1 174.546} C_DIS
LIN {X 0.184,Y -397.773,Z 593.756,A 0.000,B 0.000,C 90.000,E1 172.064} C_DIS
LIN {X -0.061,Y -397.450,Z 593.740,A 0.000,B 0.000,C 90.000,E1 169.285} C_DIS
LIN {X -0.053,Y -397.600,Z 593.729,A 0.000,B 0.000,C 90.000,E1 167.173} C_DIS
LIN {X 0.022,Y -398.040,Z 593.715,A 0.000,B 0.000,C 90.000,E1 164.700} C_DIS
LIN {X 0.127,Y -398.869,Z 593.699,A 0.000,B 0.000,C 90.000,E1 161.873} C_DIS
LIN {X -0.064,Y -399.729,Z 593.686,A 0.000,B 0.000,C 90.000,E1 159.444} C_DIS
LIN {X 0.052,Y -400.732,Z 593.672,A 0.000,B 0.000,C 90.000,E1 156.975} C_DIS
LIN {X 0.025,Y -401.520,Z 593.662,A 0.000,B 0.000,C 90.000,E1 155.229} C_DIS
LIN {X 0.060,Y -402.491,Z 593.651,A 0.000,B 0.000,C 90.000,E1 153.127} C_DIS
LIN {X 0.046,Y -403.261,Z 593.641,A 0.000,B 0.000,C 90.000,E1 151.385} C_DIS
LIN {X -0.012,Y -403.851,Z 593.633,A 0.000,B 0.000,C 90.000,E1 149.999} C_DIS
LIN {X -0.046,Y -404.603,Z 593.622,A 0.000,B 0.000,C 90.000,E1 147.916} C_DIS
LIN {X 0.025,Y -405.004,Z 593.612,A 0.000,B 0.000,C 90.000,E1 146.167} C_DIS
LIN {X 0.217,Y -405.430,Z 593.602,A 0.000,B 0.000,C 90.000,E1 144.402} C_DIS
LIN {X 0.098,Y -405.840,Z 593.593,A 0.000,B 0.000,C 90.000,E1 142.683} C_DIS
LIN {X 0.122,Y -406.399,Z 593.581,A 0.000,B 0.000,C 90.000,E1 140.598} C_DIS
LIN {X 0.047,Y -406.921,Z 593.570,A 0.000,B 0.000,C 90.000,E1 138.528} C_DIS
LIN {X 0.146,Y -407.180,Z 593.560,A 0.000,B 0.000,C 90.000,E1 136.782} C_DIS
LIN {X -0.224,Y -407.526,Z 593.549,A 0.000,B 0.000,C 90.000,E1 134.757} C_DIS
LIN {X -0.016,Y -407.758,Z 593.537,A 0.000,B 0.000,C 90.000,E1 132.651} C_DIS
LIN {X 0.095,Y -407.890,Z 593.527,A 0.000,B 0.000,C 90.000,E1 130.906} C_DIS
LIN {X -0.050,Y -408.014,Z 593.518,A 0.000,B 0.000,C 90.000,E1 129.197} C_DIS
LIN {X -0.028,Y -408.002,Z 593.514,A 0.000,B 0.000,C 90.000,E1 128.588} C_DIS
LIN {X -0.033,Y -415.177,Z 593.501,A 0.000,B 0.000,C 90.000,E1 126.091} C_DIS
LIN {X 0.078,Y -416.856,Z 593.497,A 0.000,B 0.000,C 90.000,E1 125.391} C_DIS
LIN {X 0.007,Y -426.571,Z 593.476,A 0.000,B 0.000,C 90.000,E1 121.671} C_DIS
LIN {X -0.008,Y -427.326,Z 593.475,A 0.000,B 0.000,C 90.000,E1 121.416} C_DIS
LIN {X -0.048,Y -427.389,Z 593.475,A 0.000,B 0.000,C 90.000,E1 121.416} C_DIS
LIN {X 0.036,Y -439.474,Z 593.471,A 0.000,B 0.000,C 90.000,E1 120.846} C_DIS
LIN {X 0.139,Y -452.683,Z 593.468,A 0.000,B 0.000,C 90.000,E1 120.207} C_DIS
LIN {X -0.205,Y -464.404,Z 593.465,A 0.000,B 0.000,C 90.000,E1 119.667} C_DIS
LIN {X 0.047,Y -472.915,Z 593.462,A 0.000,B 0.000,C 90.000,E1 119.205} C_DIS
LIN {X -0.129,Y -479.500,Z 593.460,A 0.000,B 0.000,C 90.000,E1 118.871} C_DIS
LIN {X -0.080,Y -489.195,Z 593.457,A 0.000,B 0.000,C 90.000,E1 118.309} C_DIS
LIN {X -0.288,Y -497.301,Z 593.455,A 0.000,B 0.000,C 90.000,E1 117.847} C_DIS
LIN {X -0.048,Y -504.923,Z 593.452,A 0.000,B 0.000,C 90.000,E1 117.334} C_DIS
LIN {X 0.061,Y -514.329,Z 593.448,A 0.000,B 0.000,C 90.000,E1 116.693} C_DIS
LIN {X -0.160,Y -520.415,Z 593.446,A 0.000,B 0.000,C 90.000,E1 116.283} C_DIS
LIN {X -0.141,Y -527.894,Z 593.443,A 0.000,B 0.000,C 90.000,E1 115.720} C_DIS
LIN {X -0.179,Y -535.222,Z 593.440,A 0.000,B 0.000,C 90.000,E1 115.155} C_DIS
LIN {X 0.188,Y -540.901,Z 593.437,A 0.000,B 0.000,C 90.000,E1 114.643} C_DIS
LIN {X 0.175,Y -546.537,Z 593.434,A 0.000,B 0.000,C 90.000,E1 114.155} C_DIS
LIN {X -0.108,Y -550.481,Z 593.432,A 0.000,B 0.000,C 90.000,E1 113.823} C_DIS
LIN {X 0.223,Y -555.532,Z 593.429,A 0.000,B 0.000,C 90.000,E1 113.259} C_DIS
LIN {X 0.132,Y -560.321,Z 593.426,A 0.000,B 0.000,C 90.000,E1 112.717} C_DIS
LIN {X 0.135,Y -565.408,Z 593.422,A 0.000,B 0.000,C 90.000,E1 112.025} C_DIS
LIN {X 0.064,Y -568.944,Z 593.419,A 0.000,B 0.000,C 90.000,E1 111.482} C_DIS
LIN {X -0.294,Y -573.497,Z 593.415,A 0.000,B 0.000,C 90.000,E1 110.737} C_DIS
LIN {X 0.071,Y -577.729,Z 593.411,A 0.000,B 0.000,C 90.000,E1 109.885} C_DIS
LIN {X -0.066,Y -581.578,Z 593.406,A 0.000,B 0.000,C 90.000,E1 109.087} C_DIS
LIN {X -0.172,Y -585.121,Z 593.402,A 0.000,B 0.000,C 90.000,E1 108.290} C_DIS
LIN {X 0.125,Y -588.369,Z 593.397,A 0.000,B 0.000,C 90.000,E1 107.457} C_DIS
LIN {X 0.155,Y -592.199,Z 593.391,A 0.000,B 0.000,C 90.000,E1 106.386} C_DIS
LIN {X -0.331,Y -595.754,Z 593.385,A 0.000,B 0.000,C 90.000,E1 105.371} C_DIS
LIN {X -0.200,Y -599.185,Z 593.379,A 0.000,B 0.000,C 90.000,E1 104.300} C_DIS
LIN {X 0.004,Y -604.322,Z 593.371,A 0.000,B 0.000,C 90.000,E1 102.703} C_DIS
LIN {X 0.134,Y -611.314,Z 593.359,A 0.000,B 0.000,C 90.000,E1 100.602} C_DIS
LIN {X 0.220,Y -614.657,Z 593.353,A 0.000,B 0.000,C 90.000,E1 99.557} C_DIS
LIN {X -0.257,Y -617.849,Z 593.348,A 0.000,B 0.000,C 90.000,E1 98.568} C_DIS
LIN {X -0.170,Y -620.984,Z 593.342,A 0.000,B 0.000,C 90.000,E1 97.530} C_DIS
LIN {X 0.038,Y -623.965,Z 593.336,A 0.000,B 0.000,C 90.000,E1 96.486} C_DIS
LIN {X -0.181,Y -626.014,Z 593.332,A 0.000,B 0.000,C 90.000,E1 95.739} C_DIS
LIN {X 0.016,Y -628.546,Z 593.326,A 0.000,B 0.000,C 90.000,E1 94.702} C_DIS
LIN {X -0.156,Y -630.105,Z 593.322,A 0.000,B 0.000,C 90.000,E1 93.955} C_DIS
LIN {X 0.045,Y -632.036,Z 593.316,A 0.000,B 0.000,C 90.000,E1 92.922} C_DIS
LIN {X 0.249,Y -633.644,Z 593.311,A 0.000,B 0.000,C 90.000,E1 91.892} C_DIS
LIN {X 0.122,Y -634.689,Z 593.306,A 0.000,B 0.000,C 90.000,E1 91.146} C_DIS
LIN {X -0.267,Y -635.788,Z 593.301,A 0.000,B 0.000,C 90.000,E1 90.172} C_DIS
LIN {X 0.247,Y -636.302,Z 593.297,A 0.000,B 0.000,C 90.000,E1 89.370} C_DIS
LIN {X 0.127,Y -636.589,Z 593.292,A 0.000,B 0.000,C 90.000,E1 88.625} C_DIS
LIN {X 0.029,Y -636.656,Z 593.288,A 0.000,B 0.000,C 90.000,E1 87.879} C_DIS
LIN {X 0.289,Y -636.390,Z 593.283,A 0.000,B 0.000,C 90.000,E1 86.849} C_DIS
LIN {X -0.020,Y -635.801,Z 593.277,A 0.000,B 0.000,C 90.000,E1 85.869} C_DIS
LIN {X 0.256,Y -634.921,Z 593.271,A 0.000,B 0.000,C 90.000,E1 84.837} C_DIS
LIN {X -0.329,Y -633.499,Z 593.264,A 0.000,B 0.000,C 90.000,E1 83.628} C_DIS
LIN {X -0.179,Y -632.800,Z 593.262,A 0.000,B 0.000,C 90.000,E1 83.109} C_DIS
LIN {X 0.189,Y -631.080,Z 593.256,A 0.000,B 0.000,C 90.000,E1 82.064} C_DIS
LIN {X 0.027,Y -629.626,Z 593.252,A 0.000,B 0.000,C 90.000,E1 81.319} C_DIS
LIN {X -0.267,Y -627.449,Z 593.246,A 0.000,B 0.000,C 90.000,E1 80.330} C_DIS
LIN {X 0.026,Y -625.120,Z 593.241,A 0.000,B 0.000,C 90.000,E1 79.285} C_DIS
LIN {X -0.024,Y -621.216,Z 593.232,A 0.000,B 0.000,C 90.000,E1 77.757} C_DIS
LIN {X -0.073,Y -619.076,Z 593.228,A 0.000,B 0.000,C 90.000,E1 76.992} C_DIS
LIN {X 0.226,Y -616.035,Z 593.222,A 0.000,B 0.000,C 90.000,E1 75.936} C_DIS
LIN {X -0.121,Y -612.788,Z 593.216,A 0.000,B 0.000,C 90.000,E1 74.936} C_DIS
LIN {X -0.101,Y -610.169,Z 593.212,A 0.000,B 0.000,C 90.000,E1 74.157} C_DIS
LIN {X -0.105,Y -607.249,Z 593.208,A 0.000,B 0.000,C 90.000,E1 73.378} C_DIS
LIN {X 0.168,Y -602.916,Z 593.202,A 0.000,B 0.000,C 90.000,E1 72.308} C_DIS
LIN {X 0.323,Y -600.009,Z 593.198,A 0.000,B 0.000,C 90.000,E1 71.638} C_DIS
LIN {X 0.153,Y -595.538,Z 593.193,A 0.000,B 0.000,C 90.000,E1 70.732} C_DIS
LIN {X 0.187,Y -591.417,Z 593.189,A 0.000,B 0.000,C 90.000,E1 69.934} C_DIS
LIN {X 0.079,Y -586.960,Z 593.184,A 0.000,B 0.000,C 90.000,E1 69.156} C_DIS
LIN {X -0.061,Y -582.963,Z 593.181,A 0.000,B 0.000,C 90.000,E1 68.518} C_DIS
LIN {X -0.079,Y -578.528,Z 593.177,A 0.000,B 0.000,C 90.000,E1 67.847} C_DIS
LIN {X 0.198,Y -573.836,Z 593.173,A 0.000,B 0.000,C 90.000,E1 67.177} C_DIS
LIN {X -0.056,Y -569.599,Z 593.170,A 0.000,B 0.000,C 90.000,E1 66.666} C_DIS
LIN {X 0.115,Y -564.893,Z 593.167,A 0.000,B 0.000,C 90.000,E1 66.102} C_DIS
LIN {X 0.301,Y -559.836,Z 593.164,A 0.000,B 0.000,C 90.000,E1 65.537} C_DIS
LIN {X -0.098,Y -554.485,Z 593.161,A 0.000,B 0.000,C 90.000,E1 65.049} C_DIS
LIN {X 0.022,Y -548.763,Z 593.159,A 0.000,B 0.000,C 90.000,E1 64.537} C_DIS
LIN {X -0.160,Y -544.295,Z 593.157,A 0.000,B 0.000,C 90.000,E1 64.204} C_DIS
LIN {X -0.086,Y -538.098,Z 593.154,A 0.000,B 0.000,C 90.000,E1 63.768} C_DIS
LIN {X 0.141,Y -531.269,Z 593.152,A 0.000,B 0.000,C 90.000,E1 63.332} C_DIS
LIN {X -0.152,Y -524.377,Z 593.150,A 0.000,B 0.000,C 90.000,E1 62.999} C_DIS
LIN {X 0.241,Y -517.483,Z 593.148,A 0.000,B 0.000,C 90.000,E1 62.615} C_DIS
LIN {X 0.163,Y -507.156,Z 593.145,A 0.000,B 0.000,C 90.000,E1 62.153} C_DIS
LIN {X -0.217,Y -491.696,Z 593.142,A 0.000,B 0.000,C 90.000,E1 61.513} C_DIS
LIN {X -0.128,Y -469.391,Z 593.136,A 0.000,B 0.000,C 90.000,E1 60.511} C_DIS
LIN {X -0.137,Y -456.112,Z 593.133,A 0.000,B 0.000,C 90.000,E1 59.871} C_DIS
LIN {X -0.034,Y -449.947,Z 593.131,A 0.000,B 0.000,C 90.000,E1 59.537} C_DIS
LIN {X -0.078,Y -449.861,Z 593.131,A 0.000,B 0.000,C 90.000,E1 59.537} C_DIS
LIN {X 0.065,Y -444.114,Z 593.114,A 0.000,B 0.000,C 90.000,E1 56.580} C_DIS
LIN {X 0.107,Y -441.691,Z 593.109,A 0.000,B 0.000,C 90.000,E1 55.595} C_DIS
LIN {X -0.061,Y -433.040,Z 593.087,A 0.000,B 0.000,C 90.000,E1 51.662} C_DIS
LIN {X 0.241,Y -433.074,Z 593.086,A 0.000,B 0.000,C 90.000,E1 51.457} C_DIS
LIN {X 0.040,Y -434.303,Z 593.078,A 0.000,B 0.000,C 90.000,E1 49.989} C_DIS
LIN {X 0.104,Y -435.682,Z 593.069,A 0.000,B 0.000,C 90.000,E1 48.324} C_DIS
LIN {X -0.230,Y -437.576,Z 593.056,A 0.000,B 0.000,C 90.000,E1 46.053} C_DIS
LIN {X 0.135,Y -439.191,Z 593.045,A 0.000,B 0.000,C 90.000,E1 44.028} C_DIS
LIN {X -0.022,Y -440.073,Z 593.037,A 0.000,B 0.000,C 90.000,E1 42.732} C_DIS
LIN {X -0.143,Y -440.799,Z 593.030,A 0.000,B 0.000,C 90.000,E1 41.434} C_DIS
LIN {X 0.042,Y -441.536,Z 593.021,A 0.000,B 0.000,C 90.000,E1 39.769} C_DIS
LIN {X -0.044,Y -442.152,Z 593.012,A 0.000,B 0.000,C 90.000,E1 38.141} C_DIS
LIN {X -0.040,Y -442.598,Z 593.003,A 0.000,B 0.000,C 90.000,E1 36.503} C_DIS
LIN {X 0.034,Y -442.822,Z 592.996,A 0.000,B 0.000,C 90.000,E1 35.185} C_DIS
LIN {X 0.118,Y -442.922,Z 592.988,A 0.000,B 0.000,C 90.000,E1 33.865} C_DIS
LIN {X -0.071,Y -443.004,Z 592.977,A 0.000,B 0.000,C 90.000,E1 31.926} C_DIS
LIN {X 0.196,Y -443.055,Z 592.968,A 0.000,B 0.000,C 90.000,E1 30.256} C_DIS
LIN {X 0.085,Y -443.154,Z 592.957,A 0.000,B 0.000,C 90.000,E1 28.309} C_DIS
LIN {X -0.021,Y -443.326,Z 592.946,A 0.000,B 0.000,C 90.000,E1 26.360} C_DIS
LIN {X 0.069,Y -443.572,Z 592.936,A 0.000,B 0.000,C 90.000,E1 24.387} C_DIS
LIN {X -0.200,Y -443.883,Z 592.925,A 0.000,B 0.000,C 90.000,E1 22.461} C_DIS
LIN {X -0.051,Y -444.298,Z 592.914,A 0.000,B 0.000,C 90.000,E1 20.482} C_DIS
LIN {X -0.068,Y -444.892,Z 592.899,A 0.000,B 0.000,C 90.000,E1 17.873} C_DIS
LIN {X 0.077,Y -445.498,Z 592.888,A 0.000,B 0.000,C 90.000,E1 15.898} C_DIS
LIN {X 0.024,Y -446.577,Z 592.874,A 0.000,B 0.000,C 90.000,E1 13.300} C_DIS
LIN {X -0.099,Y -448.040,Z 592.859,A 0.000,B 0.000,C 90.000,E1 10.715} C_DIS
LIN {X 0.073,Y -449.273,Z 592.849,A 0.000,B 0.000,C 90.000,E1 8.746} C_DIS
LIN {X -0.080,Y -451.506,Z 592.833,A 0.000,B 0.000,C 90.000,E1 5.853} C_DIS
LIN {X -0.048,Y -453.879,Z 592.818,A 0.000,B 0.000,C 90.000,E1 3.269} C_DIS
LIN {X -0.144,Y -456.267,Z 592.806,A 0.000,B 0.000,C 90.000,E1 1.031} C_DIS
LIN {X -0.169,Y -458.944,Z 592.794,A 0.000,B 0.000,C 90.000,E1 358.854} C_DIS
LIN {X 0.079,Y -462.503,Z 592.779,A 0.000,B 0.000,C 90.000,E1 356.274} C_DIS
LIN {X -0.212,Y -465.822,Z 592.767,A 0.000,B 0.000,C 90.000,E1 354.090} C_DIS
LIN {X -0.127,Y -468.780,Z 592.757,A 0.000,B 0.000,C 90.000,E1 352.186} C_DIS
LIN {X -0.087,Y -472.200,Z 592.744,A 0.000,B 0.000,C 90.000,E1 349.982} C_DIS
LIN {X -0.100,Y -476.728,Z 592.729,A 0.000,B 0.000,C 90.000,E1 347.173} C_DIS
LIN {X 0.127,Y -479.939,Z 592.718,A 0.000,B 0.000,C 90.000,E1 345.283} C_DIS
LIN {X -0.043,Y -483.385,Z 592.708,A 0.000,B 0.000,C 90.000,E1 343.449} C_DIS
LIN {X -0.198,Y -485.119,Z 592.703,A 0.000,B 0.000,C 90.000,E1 342.543} C_DIS
LIN {X 0.041,Y -489.229,Z 592.691,A 0.000,B 0.000,C 90.000,E1 340.369} C_DIS
LIN {X 0.015,Y -492.183,Z 592.683,A 0.000,B 0.000,C 90.000,E1 338.847} C_DIS
LIN {X -0.239,Y -494.891,Z 592.674,A 0.000,B 0.000,C 90.000,E1 337.358} C_DIS
LIN {X 0.212,Y -497.512,Z 592.666,A 0.000,B 0.000,C 90.000,E1 335.793} C_DIS
LIN {X -0.071,Y -499.006,Z 592.661,A 0.000,B 0.000,C 90.000,E1 334.921} C_DIS
LIN {X 0.219,Y -501.377,Z 592.652,A 0.000,B 0.000,C 90.000,E1 333.384} C_DIS
LIN {X -0.270,Y -504.093,Z 592.642,A 0.000,B 0.000,C 90.000,E1 331.641} C_DIS
LIN {X -0.030,Y -505.521,Z 592.637,A 0.000,B 0.000,C 90.000,E1 330.717} C_DIS
LIN {X -0.195,Y -508.259,Z 592.627,A 0.000,B 0.000,C 90.000,E1 328.948} C_DIS
LIN {X 0.131,Y -511.675,Z 592.616,A 0.000,B 0.000,C 90.000,E1 326.834} C_DIS
LIN {X -0.225,Y -514.791,Z 592.606,A 0.000,B 0.000,C 90.000,E1 325.102} C_DIS
LIN {X -0.216,Y -518.100,Z 592.596,A 0.000,B 0.000,C 90.000,E1 323.336} C_DIS
LIN {X 0.018,Y -519.775,Z 592.591,A 0.000,B 0.000,C 90.000,E1 322.431} C_DIS
LIN {X 0.085,Y -526.498,Z 592.574,A 0.000,B 0.000,C 90.000,E1 319.218} C_DIS
LIN {X -0.071,Y -529.076,Z 592.569,A 0.000,B 0.000,C 90.000,E1 318.366} C_DIS
LIN {X -0.104,Y -530.249,Z 592.567,A 0.000,B 0.000,C 90.000,E1 318.081} C_DIS
LIN {X 0.200,Y -533.416,Z 592.564,A 0.000,B 0.000,C 90.000,E1 317.472} C_DIS
LIN {X 0.076,Y -535.456,Z 592.562,A 0.000,B 0.000,C 90.000,E1 317.187} C_DIS
LIN {X 0.024,Y -539.469,Z 592.560,A 0.000,B 0.000,C 90.000,E1 316.743} C_DIS
LIN {X -0.146,Y -544.303,Z 592.557,A 0.000,B 0.000,C 90.000,E1 316.296} C_DIS
LIN {X -0.248,Y -550.195,Z 592.554,A 0.000,B 0.000,C 90.000,E1 315.810} C_DIS
LIN {X -0.030,Y -565.002,Z 592.548,A 0.000,B 0.000,C 90.000,E1 314.676} C_DIS
LIN {X 0.092,Y -586.822,Z 592.539,A 0.000,B 0.000,C 90.000,E1 313.056} C_DIS
LIN {X 0.006,Y -594.050,Z 592.536,A 0.000,B 0.000,C 90.000,E1 312.528} C_DIS
LIN {X 0.200,Y -602.404,Z 592.533,A 0.000,B 0.000,C 90.000,E1 311.838} C_DIS
LIN {X -0.073,Y -608.897,Z 592.529,A 0.000,B 0.000,C 90.000,E1 311.272} C_DIS
LIN {X -0.028,Y -612.723,Z 592.527,A 0.000,B 0.000,C 90.000,E1 310.906} C_DIS
LIN {X -0.093,Y -617.542,Z 592.525,A 0.000,B 0.000,C 90.000,E1 310.415} C_DIS
LIN {X -0.080,Y -622.113,Z 592.522,A 0.000,B 0.000,C 90.000,E1 309.930} C_DIS
LIN {X 0.071,Y -627.724,Z 592.518,A 0.000,B 0.000,C 90.000,E1 309.277} C_DIS
LIN {X -0.226,Y -633.129,Z 592.515,A 0.000,B 0.000,C 90.000,E1 308.669} C_DIS
LIN {X -0.436,Y -640.268,Z 592.510,A 0.000,B 0.000,C 90.000,E1 307.810} C_DIS
LIN {X -0.121,Y -645.807,Z 592.506,A 0.000,B 0.000,C 90.000,E1 307.030} C_DIS
LIN {X -0.198,Y -648.488,Z 592.504,A 0.000,B 0.000,C 90.000,E1 306.664} C_DIS
LIN {X -0.239,Y -651.767,Z 592.501,A 0.000,B 0.000,C 90.000,E1 306.171} C_DIS
LIN {X 0.230,Y -655.578,Z 592.497,A 0.000,B 0.000,C 90.000,E1 305.518} C_DIS
LIN {X 0.237,Y -658.369,Z 592.495,A 0.000,B 0.000,C 90.000,E1 305.025} C_DIS
LIN {X -0.180,Y -662.080,Z 592.491,A 0.000,B 0.000,C 90.000,E1 304.326} C_DIS
LIN {X -0.017,Y -665.493,Z 592.487,A 0.000,B 0.000,C 90.000,E1 303.579} C_DIS
LIN {X 0.183,Y -668.628,Z 592.483,A 0.000,B 0.000,C 90.000,E1 302.832} C_DIS
LIN {X 0.004,Y -672.502,Z 592.477,A 0.000,B 0.000,C 90.000,E1 301.878} C_DIS
LIN {X 0.042,Y -677.113,Z 592.470,A 0.000,B 0.000,C 90.000,E1 300.669} C_DIS
LIN {X 0.148,Y -681.467,Z 592.464,A 0.000,B 0.000,C 90.000,E1 299.461} C_DIS
LIN {X 0.369,Y -684.725,Z 592.458,A 0.000,B 0.000,C 90.000,E1 298.487} C_DIS
LIN {X -0.291,Y -687.737,Z 592.453,A 0.000,B 0.000,C 90.000,E1 297.590} C_DIS
LIN {X -0.219,Y -689.884,Z 592.449,A 0.000,B 0.000,C 90.000,E1 296.873} C_DIS
LIN {X -0.133,Y -691.343,Z 592.445,A 0.000,B 0.000,C 90.000,E1 296.155} C_DIS
LIN {X 0.044,Y -691.220,Z 592.443,A 0.000,B 0.000,C 90.000,E1 295.668} C_DIS
LIN {X 0.285,Y -691.024,Z 592.441,A 0.000,B 0.000,C 90.000,E1 295.412} C_DIS
LIN {X -0.100,Y -690.161,Z 592.440,A 0.000,B 0.000,C 90.000,E1 295.207} C_DIS
LIN {X 0.137,Y -689.126,Z 592.439,A 0.000,B 0.000,C 90.000,E1 294.951} C_DIS
LIN {X 0.082,Y -687.931,Z 592.437,A 0.000,B 0.000,C 90.000,E1 294.719} C_DIS
LIN {X 0.198,Y -686.864,Z 592.437,A 0.000,B 0.000,C 90.000,E1 294.591} C_DIS
LIN {X 0.321,Y -682.345,Z 592.435,A 0.000,B 0.000,C 90.000,E1 294.259} C_DIS
LIN {X 0.163,Y -680.971,Z 592.434,A 0.000,B 0.000,C 90.000,E1 294.155} C_DIS
LIN {X -0.251,Y -679.001,Z 592.434,A 0.000,B 0.000,C 90.000,E1 294.079} C_DIS
LIN {X -0.152,Y -674.251,Z 592.433,A 0.000,B 0.000,C 90.000,E1 293.898} C_DIS
LIN {X -0.015,Y -670.451,Z 592.432,A 0.000,B 0.000,C 90.000,E1 293.770} C_DIS
LIN {X 0.318,Y -666.113,Z 592.432,A 0.000,B 0.000,C 90.000,E1 293.643} C_DIS
LIN {X -0.183,Y -659.564,Z 592.431,A 0.000,B 0.000,C 90.000,E1 293.567} C_DIS
LIN {X 0.169,Y -642.073,Z 592.429,A 0.000,B 0.000,C 90.000,E1 293.259} C_DIS
LIN {X -0.031,Y -632.187,Z 592.428,A 0.000,B 0.000,C 90.000,E1 293.078} C_DIS
LIN {X 0.132,Y -622.409,Z 592.427,A 0.000,B 0.000,C 90.000,E1 292.823} C_DIS
LIN {X -0.062,Y -609.083,Z 592.425,A 0.000,B 0.000,C 90.000,E1 292.461} C_DIS
LIN {X -0.113,Y -579.791,Z 592.420,A 0.000,B 0.000,C 90.000,E1 291.535} C_DIS
LIN {X -0.245,Y -571.068,Z 592.418,A 0.000,B 0.000,C 90.000,E1 291.280} C_DIS
LIN {X -0.072,Y -565.338,Z 592.417,A 0.000,B 0.000,C 90.000,E1 291.046} C_DIS
LIN {X 0.199,Y -561.397,Z 592.416,A 0.000,B 0.000,C 90.000,E1 290.791} C_DIS
LIN {X 0.142,Y -561.335,Z 592.416,A 0.000,B 0.000,C 90.000,E1 290.791} C_DIS
LIN {X 0.168,Y -560.214,Z 592.415,A 0.000,B 0.000,C 90.000,E1 290.610} C_DIS
LIN {X -0.181,Y -559.612,Z 592.412,A 0.000,B 0.000,C 90.000,E1 290.248} C_DIS
LIN {X -0.119,Y -559.531,Z 592.404,A 0.000,B 0.000,C 90.000,E1 288.671} C_DIS
LIN {X -0.325,Y -559.292,Z 592.398,A 0.000,B 0.000,C 90.000,E1 287.583} C_DIS
LIN {X 0.132,Y -558.812,Z 592.390,A 0.000,B 0.000,C 90.000,E1 286.150} C_DIS
LIN {X 0.037,Y -558.171,Z 592.382,A 0.000,B 0.000,C 90.000,E1 284.773} C_DIS
LIN {X -0.086,Y -557.330,Z 592.373,A 0.000,B 0.000,C 90.000,E1 283.119} C_DIS
LIN {X -0.218,Y -556.205,Z 592.362,A 0.000,B 0.000,C 90.000,E1 281.186} C_DIS
LIN {X 0.065,Y -555.130,Z 592.351,A 0.000,B 0.000,C 90.000,E1 279.208} C_DIS
LIN {X 0.063,Y -554.424,Z 592.344,A 0.000,B 0.000,C 90.000,E1 277.814} C_DIS
LIN {X 0.134,Y -553.479,Z 592.333,A 0.000,B 0.000,C 90.000,E1 275.853} C_DIS
LIN {X 0.127,Y -552.721,Z 592.322,A 0.000,B 0.000,C 90.000,E1 273.898} C_DIS
LIN {X -0.025,Y -552.237,Z 592.312,A 0.000,B 0.000,C 90.000,E1 272.236} C_DIS
LIN {X -0.183,Y -551.897,Z 592.303,A 0.000,B 0.000,C 90.000,E1 270.573} C_DIS
LIN {X 0.251,Y -551.236,Z 592.292,A 0.000,B 0.000,C 90.000,E1 268.568} C_DIS
LIN {X 0.063,Y -550.534,Z 592.283,A 0.000,B 0.000,C 90.000,E1 266.906} C_DIS
LIN {X -0.158,Y -549.909,Z 592.275,A 0.000,B 0.000,C 90.000,E1 265.527} C_DIS
LIN {X 0.159,Y -549.154,Z 592.267,A 0.000,B 0.000,C 90.000,E1 264.090} C_DIS
LIN {X -0.126,Y -548.384,Z 592.261,A 0.000,B 0.000,C 90.000,E1 262.996} C_DIS
LIN {X -0.252,Y -547.225,Z 592.253,A 0.000,B 0.000,C 90.000,E1 261.602} C_DIS
LIN {X 0.054,Y -546.161,Z 592.247,A 0.000,B 0.000,C 90.000,E1 260.443} C_DIS
LIN {X -0.016,Y -544.532,Z 592.238,A 0.000,B 0.000,C 90.000,E1 258.757} C_DIS
LIN {X -0.107,Y -543.180,Z 592.230,A 0.000,B 0.000,C 90.000,E1 257.353} C_DIS
LIN {X 0.259,Y -540.809,Z 592.217,A 0.000,B 0.000,C 90.000,E1 255.046} C_DIS
LIN {X -0.088,Y -539.123,Z 592.208,A 0.000,B 0.000,C 90.000,E1 253.378} C_DIS
LIN {X 0.199,Y -537.210,Z 592.198,A 0.000,B 0.000,C 90.000,E1 251.638} C_DIS
LIN {X 0.155,Y -536.160,Z 592.193,A 0.000,B 0.000,C 90.000,E1 250.786} C_DIS
LIN {X 0.125,Y -534.529,Z 592.187,A 0.000,B 0.000,C 90.000,E1 249.645} C_DIS
LIN {X 0.238,Y -533.141,Z 592.182,A 0.000,B 0.000,C 90.000,E1 248.773} C_DIS
LIN {X 0.041,Y -530.484,Z 592.174,A 0.000,B 0.000,C 90.000,E1 247.358} C_DIS
LIN {X 0.174,Y -527.023,Z 592.165,A 0.000,B 0.000,C 90.000,E1 245.613} C_DIS
LIN {X 0.121,Y -524.602,Z 592.158,A 0.000,B 0.000,C 90.000,E1 244.460} C_DIS
LIN {X 0.042,Y -522.144,Z 592.152,A 0.000,B 0.000,C 90.000,E1 243.307} C_DIS
LIN {X 0.056,Y -518.768,Z 592.144,A 0.000,B 0.000,C 90.000,E1 241.847} C_DIS
LIN {X 0.126,Y -515.935,Z 592.137,A 0.000,B 0.000,C 90.000,E1 240.667} C_DIS
LIN {X 0.048,Y -510.616,Z 592.126,A 0.000,B 0.000,C 90.000,E1 238.614} C_DIS
LIN {X 0.150,Y -506.888,Z 592.117,A 0.000,B 0.000,C 90.000,E1 237.120} C_DIS
LIN {X 0.261,Y -504.476,Z 592.112,A 0.000,B 0.000,C 90.000,E1 236.215} C_DIS
LIN {X -0.054,Y -501.041,Z 592.106,A 0.000,B 0.000,C 90.000,E1 235.055} C_DIS
LIN {X 0.043,Y -492.762,Z 592.089,A 0.000,B 0.000,C 90.000,E1 232.029} C_DIS
LIN {X -0.026,Y -488.702,Z 592.081,A 0.000,B 0.000,C 90.000,E1 230.517} C_DIS
LIN {X -0.242,Y -484.728,Z 592.072,A 0.000,B 0.000,C 90.000,E1 229.013} C_DIS
LIN {X 0.042,Y -479.319,Z 592.060,A 0.000,B 0.000,C 90.000,E1 226.824} C_DIS
LIN {X 0.068,Y -474.819,Z 592.050,A 0.000,B 0.000,C 90.000,E1 224.960} C_DIS
LIN {X 0.137,Y -471.971,Z 592.043,A 0.000,B 0.000,C 90.000,E1 223.704} C_DIS
LIN {X 0.003,Y -467.576,Z 592.032,A 0.000,B 0.000,C 90.000,E1 221.838} C_DIS
LIN {X 0.065,Y -464.111,Z 592.024,A 0.000,B 0.000,C 90.000,E1 220.253} C_DIS
LIN {X -0.197,Y -460.084,Z 592.013,A 0.000,B 0.000,C 90.000,E1 218.382} C_DIS
LIN {X 0.051,Y -457.425,Z 592.006,A 0.000,B 0.000,C 90.000,E1 217.076} C_DIS
LIN {X 0.066,Y -453.534,Z 591.995,A 0.000,B 0.000,C 90.000,E1 215.152} C_DIS
LIN {X 0.178,Y -449.197,Z 591.983,A 0.000,B 0.000,C 90.000,E1 212.880} C_DIS
LIN {X -0.172,Y -444.005,Z 591.967,A 0.000,B 0.000,C 90.000,E1 210.001} C_DIS
LIN {X -0.194,Y -439.272,Z 591.952,A 0.000,B 0.000,C 90.000,E1 207.385} C_DIS
LIN {X -0.048,Y -436.393,Z 591.943,A 0.000,B 0.000,C 90.000,E1 205.720} C_DIS
LIN {X 0.073,Y -432.991,Z 591.932,A 0.000,B 0.000,C 90.000,E1 203.718} C_DIS
LIN {X 0.135,Y -428.699,Z 591.917,A 0.000,B 0.000,C 90.000,E1 201.046} C_DIS
LIN {X 0.146,Y -424.580,Z 591.902,A 0.000,B 0.000,C 90.000,E1 198.362} C_DIS
LIN {X 0.156,Y -420.821,Z 591.887,A 0.000,B 0.000,C 90.000,E1 195.662} C_DIS
LIN {X 0.204,Y -419.057,Z 591.880,A 0.000,B 0.000,C 90.000,E1 194.300} C_DIS
LIN {X 0.125,Y -417.116,Z 591.872,A 0.000,B 0.000,C 90.000,E1 192.952} C_DIS
LIN {X -0.162,Y -413.631,Z 591.859,A 0.000,B 0.000,C 90.000,E1 190.602} C_DIS
LIN {X 0.136,Y -410.177,Z 591.844,A 0.000,B 0.000,C 90.000,E1 187.814} C_DIS
LIN {X 0.182,Y -408.547,Z 591.836,A 0.000,B 0.000,C 90.000,E1 186.429} C_DIS
LIN {X 0.082,Y -404.717,Z 591.819,A 0.000,B 0.000,C 90.000,E1 183.326} C_DIS
LIN {X 0.181,Y -401.551,Z 591.799,A 0.000,B 0.000,C 90.000,E1 179.828} C_DIS
LIN {X -0.188,Y -399.474,Z 591.782,A 0.000,B 0.000,C 90.000,E1 176.731} C_DIS
LIN {X -0.005,Y -398.682,Z 591.772,A 0.000,B 0.000,C 90.000,E1 174.951} C_DIS
LIN {X 0.147,Y -397.966,Z 591.758,A 0.000,B 0.000,C 90.000,E1 172.470} C_DIS
LIN {X -0.089,Y -397.554,Z 591.743,A 0.000,B 0.000,C 90.000,E1 169.690} C_DIS
LIN {X -0.100,Y -397.712,Z 591.729,A 0.000,B 0.000,C 90.000,E1 167.229} C_DIS
LIN {X -0.016,Y -398.149,Z 591.715,A 0.000,B 0.000,C 90.000,E1 164.755} C_DIS
LIN {X -0.027,Y -398.979,Z 591.700,A 0.000,B 0.000,C 90.000,E1 161.945} C_DIS
LIN {X 0.070,Y -399.717,Z 591.688,A 0.000,B 0.000,C 90.000,E1 159.826} C_DIS
LIN {X 0.097,Y -400.534,Z 591.676,A 0.000,B 0.000,C 90.000,E1 157.720} C_DIS
LIN {X 0.069,Y -401.363,Z 591.667,A 0.000,B 0.000,C 90.000,E1 155.973} C_DIS
LIN {X -0.069,Y -402.332,Z 591.655,A 0.000,B 0.000,C 90.000,E1 153.896} C_DIS
LIN {X -0.083,Y -403.159,Z 591.645,A 0.000,B 0.000,C 90.000,E1 152.153} C_DIS
LIN {X 0.112,Y -403.911,Z 591.636,A 0.000,B 0.000,C 90.000,E1 150.383} C_DIS
LIN {X 0.068,Y -404.435,Z 591.628,A 0.000,B 0.000,C 90.000,E1 148.997} C_DIS
LIN {X 0.238,Y -404.914,Z 591.620,A 0.000,B 0.000,C 90.000,E1 147.582} C_DIS
LIN {X -0.024,Y -405.316,Z 591.610,A 0.000,B 0.000,C 90.000,E1 145.881} C_DIS
LIN {X 0.178,Y -405.731,Z 591.601,A 0.000,B 0.000,C 90.000,E1 144.116} C_DIS
LIN {X -0.044,Y -406.198,Z 591.589,A 0.000,B 0.000,C 90.000,E1 142.065} C_DIS
LIN {X -0.222,Y -406.649,Z 591.580,A 0.000,B 0.000,C 90.000,E1 140.356} C_DIS
LIN {X 0.018,Y -407.152,Z 591.568,A 0.000,B 0.000,C 90.000,E1 138.243} C_DIS
LIN {X 0.237,Y -407.445,Z 591.557,A 0.000,B 0.000,C 90.000,E1 136.134} C_DIS
LIN {X 0.187,Y -407.665,Z 591.549,A 0.000,B 0.000,C 90.000,E1 134.757} C_DIS
LIN {X 0.123,Y -407.885,Z 591.537,A 0.000,B 0.000,C 90.000,E1 132.690} C_DIS
LIN {X -0.062,Y -408.014,Z 591.528,A 0.000,B 0.000,C 90.000,E1 130.987} C_DIS
LIN {X -0.203,Y -408.114,Z 591.518,A 0.000,B 0.000,C 90.000,E1 129.277} C_DIS
LIN {X -0.210,Y -408.157,Z 591.514,A 0.000,B 0.000,C 90.000,E1 128.543} C_DIS
LIN {X 0.059,Y -414.995,Z 591.501,A 0.000,B 0.000,C 90.000,E1 126.137} C_DIS
LIN {X -0.012,Y -415.944,Z 591.499,A 0.000,B 0.000,C 90.000,E1 125.804} C_DIS
LIN {X -0.131,Y -425.434,Z 591.478,A 0.000,B 0.000,C 90.000,E1 122.084} C_DIS
LIN {X 0.044,Y -428.156,Z 591.473,A 0.000,B 0.000,C 90.000,E1 121.131} C_DIS
LIN {X 0.006,Y -428.217,Z 591.473,A 0.000,B 0.000,C 90.000,E1 121.131} C_DIS
LIN {X -0.079,Y -440.199,Z 591.470,A 0.000,B 0.000,C 90.000,E1 120.590} C_DIS
LIN {X 0.135,Y -450.674,Z 591.467,A 0.000,B 0.000,C 90.000,E1 120.079} C_DIS
LIN {X -0.158,Y -457.341,Z 591.465,A 0.000,B 0.000,C 90.000,E1 119.795} C_DIS
LIN {X 0.077,Y -472.630,Z 591.461,A 0.000,B 0.000,C 90.000,E1 118.999} C_DIS
LIN {X 0.036,Y -480.870,Z 591.459,A 0.000,B 0.000,C 90.000,E1 118.565} C_DIS
LIN {X -0.160,Y -490.790,Z 591.456,A 0.000,B 0.000,C 90.000,E1 118.025} C_DIS
LIN {X -0.081,Y -502.070,Z 591.452,A 0.000,B 0.000,C 90.000,E1 117.334} C_DIS
LIN {X -0.150,Y -513.160,Z 591.448,A 0.000,B 0.000,C 90.000,E1 116.616} C_DIS
LIN {X 0.099,Y -520.740,Z 591.445,A 0.000,B 0.000,C 90.000,E1 116.052} C_DIS
LIN {X 0.100,Y -525.256,Z 591.443,A 0.000,B 0.000,C 90.000,E1 115.720} C_DIS
LIN {X -0.053,Y -533.950,Z 591.439,A 0.000,B 0.000,C 90.000,E1 115.079} C_DIS
LIN {X 0.233,Y -541.081,Z 591.436,A 0.000,B 0.000,C 90.000,E1 114.463} C_DIS
LIN {X -0.064,Y -545.332,Z 591.434,A 0.000,B 0.000,C 90.000,E1 114.131} C_DIS
LIN {X 0.109,Y -550.488,Z 591.431,A 0.000,B 0.000,C 90.000,E1 113.643} C_DIS
LIN {X 0.057,Y -554.336,Z 591.429,A 0.000,B 0.000,C 90.000,E1 113.259} C_DIS
LIN {X -0.104,Y -560.053,Z 591.426,A 0.000,B 0.000,C 90.000,E1 112.642} C_DIS
LIN {X 0.132,Y -563.150,Z 591.423,A 0.000,B 0.000,C 90.000,E1 112.206} C_DIS
LIN {X 0.027,Y -564.277,Z 591.423,A 0.000,B 0.000,C 90.000,E1 112.078} C_DIS
LIN {X -0.150,Y -568.957,Z 591.419,A 0.000,B 0.000,C 90.000,E1 111.408} C_DIS
LIN {X 0.162,Y -573.805,Z 591.414,A 0.000,B 0.000,C 90.000,E1 110.556} C_DIS
LIN {X -0.011,Y -578.056,Z 591.410,A 0.000,B 0.000,C 90.000,E1 109.758} C_DIS
LIN {X 0.324,Y -582.630,Z 591.405,A 0.000,B 0.000,C 90.000,E1 108.779} C_DIS
LIN {X 0.043,Y -586.152,Z 591.400,A 0.000,B 0.000,C 90.000,E1 108.000} C_DIS
LIN {X -0.204,Y -589.327,Z 591.396,A 0.000,B 0.000,C 90.000,E1 107.221} C_DIS
LIN {X 0.005,Y -593.180,Z 591.390,A 0.000,B 0.000,C 90.000,E1 106.134} C_DIS
LIN {X 0.098,Y -596.857,Z 591.384,A 0.000,B 0.000,C 90.000,E1 105.064} C_DIS
LIN {X -0.190,Y -601.147,Z 591.376,A 0.000,B 0.000,C 90.000,E1 103.772} C_DIS
LIN {X 0.325,Y -605.543,Z 591.369,A 0.000,B 0.000,C 90.000,E1 102.411} C_DIS
LIN {X 0.148,Y -611.723,Z 591.359,A 0.000,B 0.000,C 90.000,E1 100.602} C_DIS
LIN {X -0.116,Y -614.282,Z 591.355,A 0.000,B 0.000,C 90.000,E1 99.849} C_DIS
LIN {X 0.013,Y -617.592,Z 591.349,A 0.000,B 0.000,C 90.000,E1 98.803} C_DIS
LIN {X -0.137,Y -621.544,Z 591.342,A 0.000,B 0.000,C 90.000,E1 97.530} C_DIS
LIN {X 0.079,Y -624.556,Z 591.336,A 0.000,B 0.000,C 90.000,E1 96.486} C_DIS
LIN {X -0.134,Y -626.642,Z 591.332,A 0.000,B 0.000,C 90.000,E1 95.739} C_DIS
LIN {X 0.072,Y -629.205,Z 591.326,A 0.000,B 0.000,C 90.000,E1 94.702} C_DIS
LIN {X -0.093,Y -630.803,Z 591.322,A 0.000,B 0.000,C 90.000,E1 93.955} C_DIS
LIN {X 0.118,Y -632.740,Z 591.316,A 0.000,B 0.000,C 90.000,E1 92.922} C_DIS
LIN {X -0.302,Y -634.409,Z 591.311,A 0.000,B 0.000,C 90.000,E1 91.949} C_DIS
LIN {X 0.212,Y -635.462,Z 591.307,A 0.000,B 0.000,C 90.000,E1 91.146} C_DIS
LIN {X -0.167,Y -636.526,Z 591.301,A 0.000,B 0.000,C 90.000,E1 90.172} C_DIS
LIN {X -0.282,Y -637.048,Z 591.297,A 0.000,B 0.000,C 90.000,E1 89.427} C_DIS
LIN {X 0.243,Y -637.337,Z 591.293,A 0.000,B 0.000,C 90.000,E1 88.625} C_DIS
LIN {X 0.153,Y -637.405,Z 591.288,A 0.000,B 0.000,C 90.000,E1 87.879} C_DIS
LIN {X -0.214,Y -637.111,Z 591.283,A 0.000,B 0.000,C 90.000,E1 86.906} C_DIS
LIN {X -0.302,Y -636.722,Z 591.279,A 0.000,B 0.000,C 90.000,E1 86.159} C_DIS
LIN {X 0.035,Y -635.865,Z 591.273,A 0.000,B 0.000,C 90.000,E1 85.122} C_DIS
LIN {X 0.104,Y -634.510,Z 591.266,A 0.000,B 0.000,C 90.000,E1 83.856} C_DIS
LIN {X 0.263,Y -633.873,Z 591.263,A 0.000,B 0.000,C 90.000,E1 83.337} C_DIS
LIN {X -0.062,Y -632.171,Z 591.258,A 0.000,B 0.000,C 90.000,E1 82.356} C_DIS
LIN {X -0.122,Y -630.762,Z 591.253,A 0.000,B 0.000,C 90.000,E1 81.602} C_DIS
LIN {X -0.080,Y -628.022,Z 591.246,A 0.000,B 0.000,C 90.000,E1 80.330} C_DIS
LIN {X 0.223,Y -625.603,Z 591.241,A 0.000,B 0.000,C 90.000,E1 79.285} C_DIS
LIN {X -0.216,Y -622.319,Z 591.234,A 0.000,B 0.000,C 90.000,E1 78.049} C_DIS
LIN {X 0.353,Y -620.225,Z 591.229,A 0.000,B 0.000,C 90.000,E1 77.229} C_DIS
LIN {X 0.067,Y -617.152,Z 591.224,A 0.000,B 0.000,C 90.000,E1 76.228} C_DIS
LIN {X -0.261,Y -613.881,Z 591.218,A 0.000,B 0.000,C 90.000,E1 75.227} C_DIS
LIN {X -0.229,Y -611.266,Z 591.214,A 0.000,B 0.000,C 90.000,E1 74.448} C_DIS
LIN {X 0.111,Y -607.354,Z 591.208,A 0.000,B 0.000,C 90.000,E1 73.378} C_DIS
LIN {X -0.190,Y -602.946,Z 591.202,A 0.000,B 0.000,C 90.000,E1 72.362} C_DIS
LIN {X 0.016,Y -600.589,Z 591.199,A 0.000,B 0.000,C 90.000,E1 71.819} C_DIS
LIN {X -0.196,Y -595.381,Z 591.193,A 0.000,B 0.000,C 90.000,E1 70.786} C_DIS
LIN {X -0.316,Y -591.190,Z 591.189,A 0.000,B 0.000,C 90.000,E1 70.007} C_DIS
LIN {X -0.326,Y -586.519,Z 591.184,A 0.000,B 0.000,C 90.000,E1 69.209} C_DIS
LIN {X -0.103,Y -582.258,Z 591.181,A 0.000,B 0.000,C 90.000,E1 68.518} C_DIS
LIN {X 0.132,Y -577.823,Z 591.177,A 0.000,B 0.000,C 90.000,E1 67.847} C_DIS
LIN {X -0.311,Y -574.721,Z 591.175,A 0.000,B 0.000,C 90.000,E1 67.486} C_DIS
LIN {X 0.061,Y -572.637,Z 591.173,A 0.000,B 0.000,C 90.000,E1 67.177} C_DIS
LIN {X 0.252,Y -568.183,Z 591.170,A 0.000,B 0.000,C 90.000,E1 66.613} C_DIS
LIN {X -0.081,Y -563.306,Z 591.167,A 0.000,B 0.000,C 90.000,E1 66.102} C_DIS
LIN {X -0.143,Y -558.513,Z 591.164,A 0.000,B 0.000,C 90.000,E1 65.613} C_DIS
LIN {X 0.279,Y -553.594,Z 591.162,A 0.000,B 0.000,C 90.000,E1 65.101} C_DIS
LIN {X 0.088,Y -548.260,Z 591.159,A 0.000,B 0.000,C 90.000,E1 64.665} C_DIS
LIN {X -0.044,Y -543.718,Z 591.157,A 0.000,B 0.000,C 90.000,E1 64.332} C_DIS
LIN {X 0.047,Y -537.401,Z 591.155,A 0.000,B 0.000,C 90.000,E1 63.896} C_DIS
LIN {X 0.057,Y -532.278,Z 591.153,A 0.000,B 0.000,C 90.000,E1 63.589} C_DIS
LIN {X -0.208,Y -525.447,Z 591.151,A 0.000,B 0.000,C 90.000,E1 63.256} C_DIS
LIN {X 0.243,Y -518.658,Z 591.149,A 0.000,B 0.000,C 90.000,E1 62.871} C_DIS
LIN {X 0.101,Y -511.680,Z 591.148,A 0.000,B 0.000,C 90.000,E1 62.564} C_DIS
LIN {X -0.226,Y -492.798,Z 591.143,A 0.000,B 0.000,C 90.000,E1 61.769} C_DIS
LIN {X -0.042,Y -462.273,Z 591.135,A 0.000,B 0.000,C 90.000,E1 60.383} C_DIS
LIN {X -0.090,Y -450.488,Z 591.132,A 0.000,B 0.000,C 90.000,E1 59.793} C_DIS
LIN {X -0.133,Y -450.409,Z 591.132,A 0.000,B 0.000,C 90.000,E1 59.793} C_DIS
LIN {X 0.280,Y -443.867,Z 591.114,A 0.000,B 0.000,C 90.000,E1 56.421} C_DIS
LIN {X -0.047,Y -434.058,Z 591.090,A 0.000,B 0.000,C 90.000,E1 52.190} C_DIS
LIN {X 0.222,Y -433.416,Z 591.088,A 0.000,B 0.000,C 90.000,E1 51.823} C_DIS
LIN {X -0.084,Y -433.447,Z 591.087,A 0.000,B 0.000,C 90.000,E1 51.698} C_DIS
LIN {X -0.005,Y -434.739,Z 591.079,A 0.000,B 0.000,C 90.000,E1 50.194} C_DIS
LIN {X -0.272,Y -436.451,Z 591.068,A 0.000,B 0.000,C 90.000,E1 48.243} C_DIS
LIN {X 0.035,Y -438.385,Z 591.055,A 0.000,B 0.000,C 90.000,E1 45.891} C_DIS
LIN {X -0.164,Y -439.790,Z 591.046,A 0.000,B 0.000,C 90.000,E1 44.271} C_DIS
LIN {X 0.013,Y -440.723,Z 591.039,A 0.000,B 0.000,C 90.000,E1 42.933} C_DIS
LIN {X 0.202,Y -441.452,Z 591.031,A 0.000,B 0.000,C 90.000,E1 41.595} C_DIS
LIN {X 0.104,Y -442.068,Z 591.024,A 0.000,B 0.000,C 90.000,E1 40.297} C_DIS
LIN {X 0.032,Y -442.699,Z 591.015,A 0.000,B 0.000,C 90.000,E1 38.669} C_DIS
LIN {X 0.011,Y -443.097,Z 591.008,A 0.000,B 0.000,C 90.000,E1 37.363} C_DIS
LIN {X -0.269,Y -443.411,Z 591.000,A 0.000,B 0.000,C 90.000,E1 36.091} C_DIS
LIN {X 0.125,Y -443.587,Z 590.991,A 0.000,B 0.000,C 90.000,E1 34.405} C_DIS
LIN {X 0.007,Y -443.606,Z 590.979,A 0.000,B 0.000,C 90.000,E1 32.133} C_DIS
LIN {X -0.095,Y -443.645,Z 590.969,A 0.000,B 0.000,C 90.000,E1 30.512} C_DIS
LIN {X -0.039,Y -443.655,Z 590.960,A 0.000,B 0.000,C 90.000,E1 28.871} C_DIS
LIN {X 0.106,Y -443.813,Z 590.948,A 0.000,B 0.000,C 90.000,E1 26.565} C_DIS
LIN {X 0.072,Y -444.020,Z 590.935,A 0.000,B 0.000,C 90.000,E1 24.283} C_DIS
LIN {X 0.135,Y -444.278,Z 590.926,A 0.000,B 0.000,C 90.000,E1 22.642} C_DIS
LIN {X -0.004,Y -444.710,Z 590.913,A 0.000,B 0.000,C 90.000,E1 20.375} C_DIS
LIN {X 0.003,Y -445.074,Z 590.902,A 0.000,B 0.000,C 90.000,E1 18.417} C_DIS
LIN {X 0.009,Y -445.738,Z 590.890,A 0.000,B 0.000,C 90.000,E1 16.134} C_DIS
LIN {X -0.039,Y -446.757,Z 590.875,A 0.000,B 0.000,C 90.000,E1 13.536} C_DIS
LIN {X 0.031,Y -448.353,Z 590.859,A 0.000,B 0.000,C 90.000,E1 10.602} C_DIS
LIN {X -0.034,Y -449.770,Z 590.846,A 0.000,B 0.000,C 90.000,E1 8.341} C_DIS
LIN {X 0.079,Y -451.778,Z 590.832,A 0.000,B 0.000,C 90.000,E1 5.739} C_DIS
LIN {X 0.125,Y -454.144,Z 590.818,A 0.000,B 0.000,C 90.000,E1 3.154} C_DIS
LIN {X 0.223,Y -456.868,Z 590.803,A 0.000,B 0.000,C 90.000,E1 0.573} C_DIS
LIN {X 0.026,Y -459.481,Z 590.792,A 0.000,B 0.000,C 90.000,E1 358.511} C_DIS
LIN {X 0.085,Y -462.635,Z 590.779,A 0.000,B 0.000,C 90.000,E1 356.274} C_DIS
LIN {X -0.202,Y -465.915,Z 590.767,A 0.000,B 0.000,C 90.000,E1 354.090} C_DIS
LIN {X -0.116,Y -468.874,Z 590.757,A 0.000,B 0.000,C 90.000,E1 352.186} C_DIS
LIN {X -0.073,Y -472.272,Z 590.744,A 0.000,B 0.000,C 90.000,E1 349.982} C_DIS
LIN {X -0.162,Y -475.189,Z 590.734,A 0.000,B 0.000,C 90.000,E1 348.117} C_DIS
LIN {X 0.021,Y -478.390,Z 590.724,A 0.000,B 0.000,C 90.000,E1 346.228} C_DIS
LIN {X 0.123,Y -482.831,Z 590.710,A 0.000,B 0.000,C 90.000,E1 343.740} C_DIS
LIN {X -0.178,Y -485.163,Z 590.703,A 0.000,B 0.000,C 90.000,E1 342.543} C_DIS
LIN {X 0.061,Y -489.259,Z 590.691,A 0.000,B 0.000,C 90.000,E1 340.369} C_DIS
LIN {X 0.036,Y -492.210,Z 590.683,A 0.000,B 0.000,C 90.000,E1 338.847} C_DIS
LIN {X -0.216,Y -494.940,Z 590.674,A 0.000,B 0.000,C 90.000,E1 337.358} C_DIS
LIN {X 0.235,Y -497.560,Z 590.666,A 0.000,B 0.000,C 90.000,E1 335.793} C_DIS
LIN {X 0.224,Y -499.521,Z 590.659,A 0.000,B 0.000,C 90.000,E1 334.588} C_DIS
LIN {X -0.142,Y -501.911,Z 590.651,A 0.000,B 0.000,C 90.000,E1 333.127} C_DIS
LIN {X -0.002,Y -505.612,Z 590.637,A 0.000,B 0.000,C 90.000,E1 330.717} C_DIS
LIN {X 0.161,Y -508.842,Z 590.626,A 0.000,B 0.000,C 90.000,E1 328.614} C_DIS
LIN {X 0.164,Y -511.793,Z 590.616,A 0.000,B 0.000,C 90.000,E1 326.834} C_DIS
LIN {X -0.189,Y -514.902,Z 590.606,A 0.000,B 0.000,C 90.000,E1 325.102} C_DIS
LIN {X 0.115,Y -519.329,Z 590.593,A 0.000,B 0.000,C 90.000,E1 322.718} C_DIS
LIN {X -0.094,Y -524.455,Z 590.578,A 0.000,B 0.000,C 90.000,E1 320.114} C_DIS
LIN {X 0.086,Y -527.013,Z 590.572,A 0.000,B 0.000,C 90.000,E1 318.933} C_DIS
LIN {X -0.067,Y -529.533,Z 590.567,A 0.000,B 0.000,C 90.000,E1 318.081} C_DIS
LIN {X 0.064,Y -531.636,Z 590.565,A 0.000,B 0.000,C 90.000,E1 317.634} C_DIS
LIN {X -0.355,Y -532.851,Z 590.563,A 0.000,B 0.000,C 90.000,E1 317.391} C_DIS
LIN {X 0.156,Y -535.485,Z 590.561,A 0.000,B 0.000,C 90.000,E1 316.905} C_DIS
LIN {X -0.070,Y -538.882,Z 590.558,A 0.000,B 0.000,C 90.000,E1 316.500} C_DIS
LIN {X 0.119,Y -543.144,Z 590.556,A 0.000,B 0.000,C 90.000,E1 316.053} C_DIS
LIN {X 0.303,Y -547.413,Z 590.554,A 0.000,B 0.000,C 90.000,E1 315.648} C_DIS
LIN {X 0.283,Y -555.834,Z 590.550,A 0.000,B 0.000,C 90.000,E1 315.000} C_DIS
LIN {X -0.012,Y -567.724,Z 590.545,A 0.000,B 0.000,C 90.000,E1 314.150} C_DIS
LIN {X 0.213,Y -576.625,Z 590.542,A 0.000,B 0.000,C 90.000,E1 313.461} C_DIS
LIN {X -0.040,Y -589.873,Z 590.536,A 0.000,B 0.000,C 90.000,E1 312.528} C_DIS
LIN {X -0.146,Y -596.899,Z 590.533,A 0.000,B 0.000,C 90.000,E1 312.000} C_DIS
LIN {X -0.274,Y -601.126,Z 590.531,A 0.000,B 0.000,C 90.000,E1 311.676} C_DIS
LIN {X -0.010,Y -607.726,Z 590.528,A 0.000,B 0.000,C 90.000,E1 311.067} C_DIS
LIN {X 0.047,Y -611.609,Z 590.526,A 0.000,B 0.000,C 90.000,E1 310.701} C_DIS
LIN {X -0.041,Y -616.571,Z 590.523,A 0.000,B 0.000,C 90.000,E1 310.216} C_DIS
LIN {X -0.159,Y -620.189,Z 590.521,A 0.000,B 0.000,C 90.000,E1 309.850} C_DIS
LIN {X -0.001,Y -624.800,Z 590.518,A 0.000,B 0.000,C 90.000,E1 309.322} C_DIS
LIN {X -0.364,Y -632.471,Z 590.514,A 0.000,B 0.000,C 90.000,E1 308.463} C_DIS
LIN {X 0.257,Y -639.667,Z 590.509,A 0.000,B 0.000,C 90.000,E1 307.523} C_DIS
LIN {X 0.072,Y -646.199,Z 590.504,A 0.000,B 0.000,C 90.000,E1 306.664} C_DIS
LIN {X -0.072,Y -651.206,Z 590.500,A 0.000,B 0.000,C 90.000,E1 305.931} C_DIS
LIN {X -0.096,Y -654.307,Z 590.497,A 0.000,B 0.000,C 90.000,E1 305.438} C_DIS
LIN {X -0.100,Y -657.180,Z 590.494,A 0.000,B 0.000,C 90.000,E1 304.945} C_DIS
LIN {X 0.015,Y -660.980,Z 590.490,A 0.000,B 0.000,C 90.000,E1 304.199} C_DIS
LIN {X -0.002,Y -662.790,Z 590.488,A 0.000,B 0.000,C 90.000,E1 303.833} C_DIS
LIN {X 0.168,Y -666.068,Z 590.484,A 0.000,B 0.000,C 90.000,E1 303.086} C_DIS
LIN {X 0.372,Y -669.138,Z 590.480,A 0.000,B 0.000,C 90.000,E1 302.339} C_DIS
LIN {X 0.193,Y -672.988,Z 590.474,A 0.000,B 0.000,C 90.000,E1 301.386} C_DIS
LIN {X -0.291,Y -676.711,Z 590.469,A 0.000,B 0.000,C 90.000,E1 300.463} C_DIS
LIN {X 0.202,Y -680.255,Z 590.464,A 0.000,B 0.000,C 90.000,E1 299.461} C_DIS
LIN {X 0.407,Y -683.562,Z 590.458,A 0.000,B 0.000,C 90.000,E1 298.487} C_DIS
LIN {X -0.267,Y -686.577,Z 590.453,A 0.000,B 0.000,C 90.000,E1 297.590} C_DIS
LIN {X -0.206,Y -688.710,Z 590.449,A 0.000,B 0.000,C 90.000,E1 296.873} C_DIS
LIN {X 0.255,Y -689.803,Z 590.447,A 0.000,B 0.000,C 90.000,E1 296.360} C_DIS
LIN {X -0.131,Y -690.162,Z 590.445,A 0.000,B 0.000,C 90.000,E1 296.155} C_DIS
LIN {X -0.198,Y -690.282,Z 590.444,A 0.000,B 0.000,C 90.000,E1 295.924} C_DIS
LIN {X 0.039,Y -690.188,Z 590.443,A 0.000,B 0.000,C 90.000,E1 295.668} C_DIS
LIN {X 0.276,Y -689.902,Z 590.441,A 0.000,B 0.000,C 90.000,E1 295.412} C_DIS
LIN {X -0.111,Y -689.059,Z 590.440,A 0.000,B 0.000,C 90.000,E1 295.207} C_DIS
LIN {X -0.053,Y -687.533,Z 590.438,A 0.000,B 0.000,C 90.000,E1 294.847} C_DIS
LIN {X 0.063,Y -686.747,Z 590.437,A 0.000,B 0.000,C 90.000,E1 294.719} C_DIS
LIN {X 0.176,Y -685.525,Z 590.437,A 0.000,B 0.000,C 90.000,E1 294.591} C_DIS
LIN {X 0.288,Y -683.793,Z 590.436,A 0.000,B 0.000,C 90.000,E1 294.463} C_DIS
LIN {X -0.331,Y -680.208,Z 590.434,A 0.000,B 0.000,C 90.000,E1 294.207} C_DIS
LIN {X -0.148,Y -678.063,Z 590.434,A 0.000,B 0.000,C 90.000,E1 294.079} C_DIS
LIN {X 0.207,Y -671.821,Z 590.432,A 0.000,B 0.000,C 90.000,E1 293.823} C_DIS
LIN {X 0.103,Y -669.895,Z 590.432,A 0.000,B 0.000,C 90.000,E1 293.770} C_DIS
LIN {X 0.056,Y -661.221,Z 590.431,A 0.000,B 0.000,C 90.000,E1 293.590} C_DIS
LIN {X 0.314,Y -642.415,Z 590.429,A 0.000,B 0.000,C 90.000,E1 293.259} C_DIS
LIN {X 0.117,Y -632.513,Z 590.428,A 0.000,B 0.000,C 90.000,E1 293.078} C_DIS
LIN {X -0.055,Y -619.600,Z 590.427,A 0.000,B 0.000,C 90.000,E1 292.770} C_DIS
LIN {X -0.135,Y -602.761,Z 590.424,A 0.000,B 0.000,C 90.000,E1 292.280} C_DIS
LIN {X 0.080,Y -580.190,Z 590.420,A 0.000,B 0.000,C 90.000,E1 291.535} C_DIS
LIN {X -0.068,Y -571.481,Z 590.418,A 0.000,B 0.000,C 90.000,E1 291.280} C_DIS
LIN {X 0.091,Y -565.774,Z 590.417,A 0.000,B 0.000,C 90.000,E1 291.046} C_DIS
LIN {X 0.247,Y -561.681,Z 590.416,A 0.000,B 0.000,C 90.000,E1 290.791} C_DIS
LIN {X 0.218,Y -561.639,Z 590.416,A 0.000,B 0.000,C 90.000,E1 290.791} C_DIS
LIN {X 0.125,Y -560.424,Z 590.415,A 0.000,B 0.000,C 90.000,E1 290.610} C_DIS
LIN {X -0.054,Y -559.880,Z 590.412,A 0.000,B 0.000,C 90.000,E1 290.248} C_DIS
LIN {X -0.195,Y -559.828,Z 590.404,A 0.000,B 0.000,C 90.000,E1 288.671} C_DIS
LIN {X 0.138,Y -559.591,Z 590.398,A 0.000,B 0.000,C 90.000,E1 287.528} C_DIS
LIN {X 0.221,Y -559.084,Z 590.390,A 0.000,B 0.000,C 90.000,E1 286.134} C_DIS
LIN {X -0.162,Y -558.608,Z 590.384,A 0.000,B 0.000,C 90.000,E1 285.064} C_DIS
LIN {X 0.263,Y -557.748,Z 590.374,A 0.000,B 0.000,C 90.000,E1 283.355} C_DIS
LIN {X 0.143,Y -556.623,Z 590.364,A 0.000,B 0.000,C 90.000,E1 281.422} C_DIS
LIN {X -0.108,Y -555.547,Z 590.353,A 0.000,B 0.000,C 90.000,E1 279.500} C_DIS
LIN {X 0.026,Y -554.672,Z 590.344,A 0.000,B 0.000,C 90.000,E1 277.814} C_DIS
